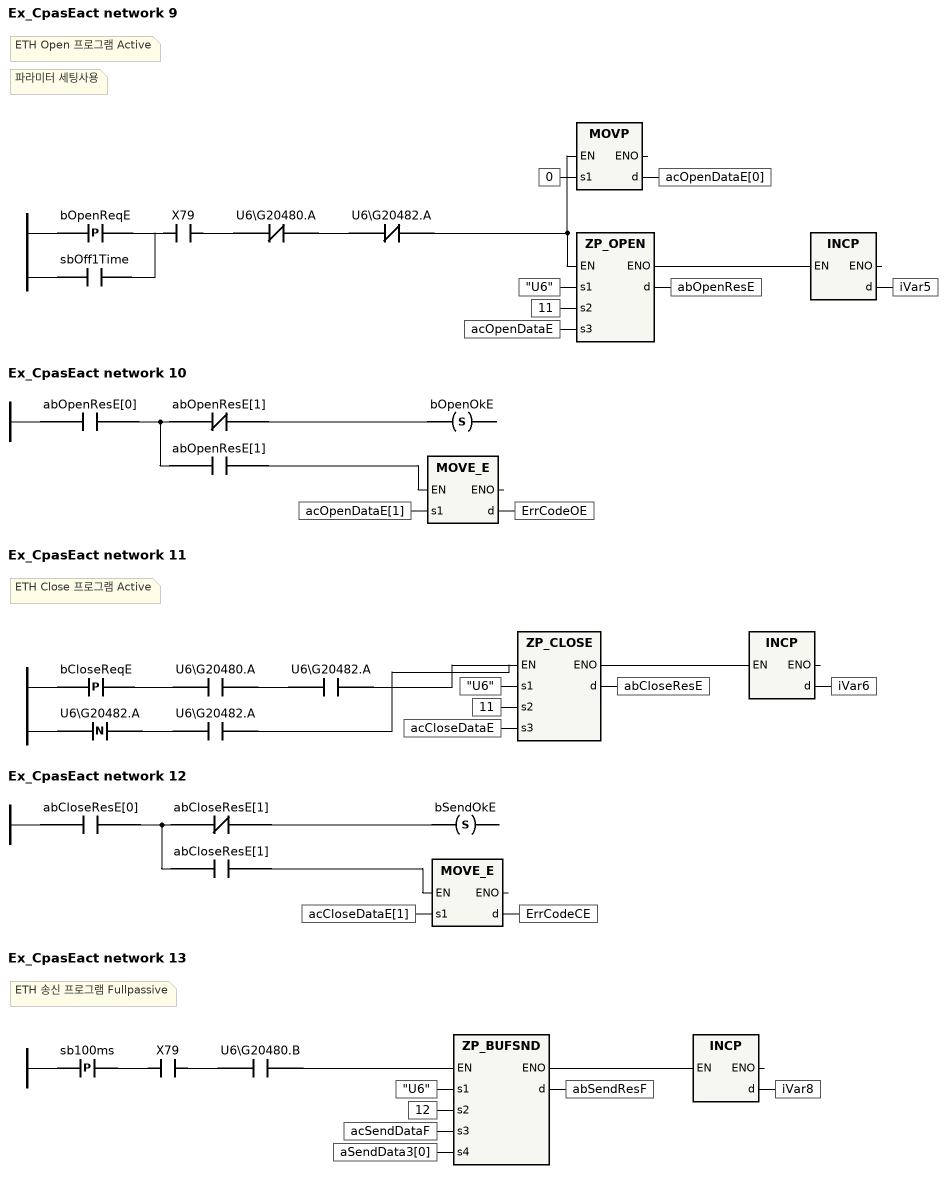
(* [picture p24: structured ladder/FBD of Ex_CpasEact, networks 9 to 13] *)
(* network 9 *)
(* ETH Open 프로그램 Active *)
(* 파라미터 세팅사용 *)
_p1 := (((LDP(TRUE, bOpenReqE) OR sbOff1Time) AND X79) AND NOT U6\G20480.A) AND NOT U6\G20482.A;
MOVP(_p1, 0, acOpenDataE[0]);
_e2 := ZP_OPEN(_p1, "U6", 11, acOpenDataE, abOpenResE);
INCP(_e2, iVar5);
(* network 10 *)
SET(abOpenResE[0] AND NOT abOpenResE[1], bOpenOkE);
MOVE_E(abOpenResE[0] AND abOpenResE[1], acOpenDataE[1], ErrCodeOE);
(* network 11 *)
(* ETH Close 프로그램 Active *)
_e1 := ZP_CLOSE((LDP(TRUE, bCloseReqE) AND U6\G20480.A AND U6\G20482.A) OR (LDF(TRUE, U6\G20482.A) AND U6\G20482.A), "U6", 11, acCloseDataE, abCloseResE);
INCP(_e1, iVar6);
(* network 12 *)
SET(abCloseResE[0] AND NOT abCloseResE[1], bSendOkE);
MOVE_E(abCloseResE[0] AND abCloseResE[1], acCloseDataE[1], ErrCodeCE);
(* network 13 *)
(* ETH 송신 프로그램 Fullpassive *)
_e1 := ZP_BUFSND(LDP(TRUE, sb100ms) AND X79 AND U6\G20480.B, "U6", 12, acSendDataF, aSendData3[0], abSendResF);
INCP(_e1, iVar8);
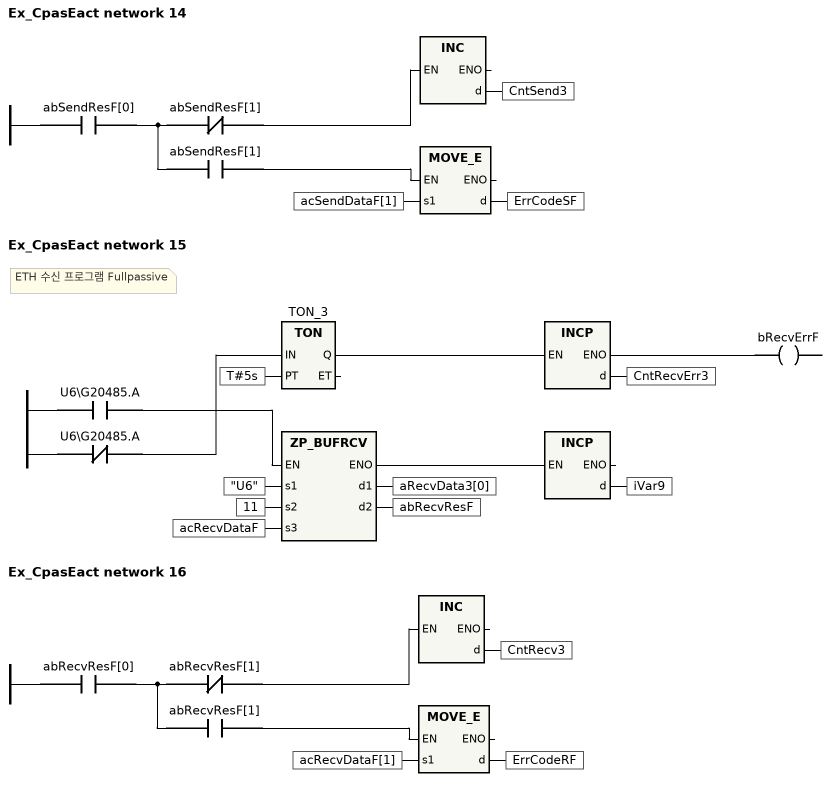
(* network 14 *)
INC(abSendResF[0] AND NOT abSendResF[1], CntSend3);
MOVE_E(abSendResF[0] AND abSendResF[1], acSendDataF[1], ErrCodeSF);
(* network 15 *)
(* ETH 수신 프로그램 Fullpassive *)
_e1 := ZP_BUFRCV(U6\G20485.A, "U6", 11, acRecvDataF, aRecvData3[0], abRecvResF);
INCP(_e1, iVar9);
TON_3(IN := NOT U6\G20485.A, PT := T#5s);
_e2 := INCP(TON_3.Q, CntRecvErr3);
bRecvErrF := _e2;
(* network 16 *)
INC(abRecvResF[0] AND NOT abRecvResF[1], CntRecv3);
MOVE_E(abRecvResF[0] AND abRecvResF[1], acRecvDataF[1], ErrCodeRF);
END_PROGRAM

PROGRAM Ex_SOCOPEN
VAR
  bOpenReqC : BOOL;
  bCsetReq : BOOL;
  bOpenReqE : BOOL;
  bOpenOkC : BOOL;
  bOpenOkE : BOOL;
  bOpenErrC : BOOL;
  bOpenErrE : BOOL;
  abOpenResC : ARRAY [0..1] OF BOOL;
  abOpenResE : ARRAY [0..1] OF BOOL;
  acOpenData : ARRAY [0..9] OF INT;
  acCsetData : ARRAY [0..4] OF INT;
  acRdCtrl : ARRAY [0..9] OF INT;
  bSendReqC : BOOL;
  bSendReqE : BOOL;
  bSendOkC : BOOL;
  bSendOkE : BOOL;
  bSendErrC : BOOL;
  bSendErrE : BOOL;
  abSendResC : ARRAY [0..1] OF BOOL;
  abSendResE : ARRAY [0..1] OF BOOL;
  abSendResF : ARRAY [0..1] OF BOOL;
  acSendDataC : ARRAY [0..1] OF INT;
  acSendDataE : ARRAY [0..1] OF INT;
  acSendDataF : ARRAY [0..1] OF INT;
  bRecvOkC : BOOL;
  bRecvOkE : BOOL;
  bRecvOkF : BOOL;
  bRecvErrC : BOOL;
  bRecvErrE : BOOL;
  bRecvErrF : BOOL;
  abRecvResC : ARRAY [0..1] OF BOOL;
  abRecvResE : ARRAY [0..1] OF BOOL;
  abRecvResF : ARRAY [0..1] OF BOOL;
  acRecvDataC : ARRAY [0..1] OF INT;
  acRecvDataE : ARRAY [0..1] OF INT;
  acRecvDataF : ARRAY [0..1] OF INT;
  bCloseReq : BOOL;
  bCloseOkC : BOOL;
  bCloseOkE : BOOL;
  bCloseErrC : BOOL;
  bCloseErrE : BOOL;
  abCloseResC : ARRAY [0..1] OF BOOL;
  abCloseResE : ARRAY [0..1] OF BOOL;
  acCloseData : ARRAY [0..1] OF INT;
  CntSend1 : INT;
  CntSend2 : INT;
  CntSend3 : INT;
  CntRecv1 : INT;
  CntRecvErr1 : INT;
  CntRecv2 : INT;
  CntRecv3 : INT;
  CntRecvErr2 : INT;
  CntRecvErr3 : INT;
  ErrCodeSC : INT;
  ErrCodeSE : INT;
  ErrCodeSF : INT;
  ErrCodeRC : INT;
  ErrCodeRE : INT;
  ErrCodeRF : INT;
  Mov4INT_1 : Mov4INT;
  Mov8INT_1 : Mov8INT;
  Mov4INT_2 : Mov4INT;
  Mov4INT_3 : Mov4INT;
  Mov4INT_4 : Mov4INT;
  Word2Bit8_1 : Word2Bit8;
  Word2Bit8_2 : Word2Bit8;
  Word2Bit8_3 : Word2Bit8;
  Word2Bit8_4 : Word2Bit8;
  Word2Bit8_5 : Word2Bit8;
  Word2Bit8_6 : Word2Bit8;
  TON_1 : TON;
  TON_2 : TON;
  TON_3 : TON;
END_VAR
(* structured ladder/FBD written out as ST: instructions are called as NAME(EN, inputs, outputs); _pN, _eN, _tN stand for wires *)
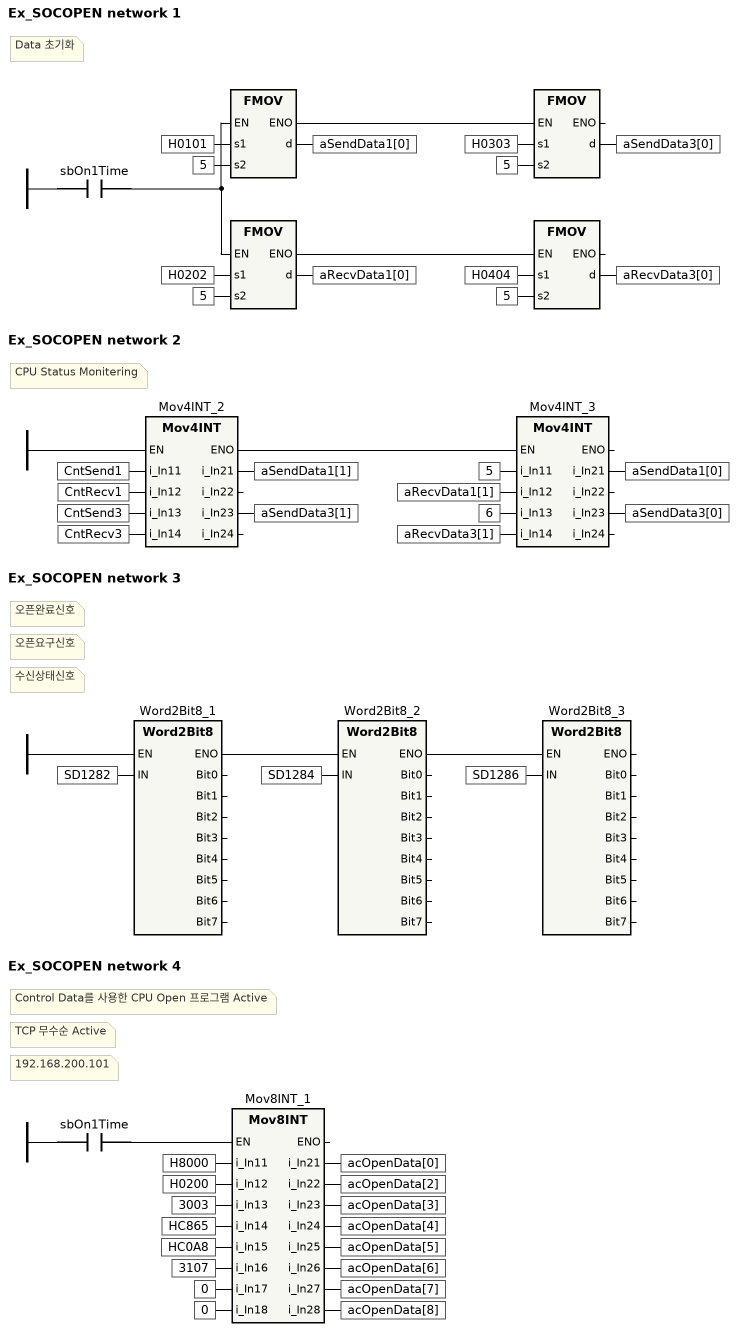
(* network 1 *)
(* Data 초기화 *)
_e1 := FMOV(sbOn1Time, H0101, 5, aSendData1[0]);
FMOV(_e1, H0303, 5, aSendData3[0]);
_e2 := FMOV(sbOn1Time, H0202, 5, aRecvData1[0]);
FMOV(_e2, H0404, 5, aRecvData3[0]);
(* network 2 *)
(* CPU Status Monitering *)
Mov4INT_2(EN := TRUE, i_In11 := CntSend1, i_In12 := CntRecv1, i_In13 := CntSend3, i_In14 := CntRecv3, i_In21 => aSendData1[1], i_In23 => aSendData3[1]);
Mov4INT_3(EN := Mov4INT_2.ENO, i_In11 := 5, i_In12 := aRecvData1[1], i_In13 := 6, i_In14 := aRecvData3[1], i_In21 => aSendData1[0], i_In23 => aSendData3[0]);
(* network 3 *)
(* 오픈완료신호 *)
(* 오픈요구신호 *)
(* 수신상태신호 *)
Word2Bit8_1(EN := TRUE, IN := SD1282);
Word2Bit8_2(EN := Word2Bit8_1.ENO, IN := SD1284);
Word2Bit8_3(EN := Word2Bit8_2.ENO, IN := SD1286);
(* network 4 *)
(* Control Data를 사용한 CPU Open 프로그램 Active *)
(* TCP 무수순 Active *)
(* 192.168.200.101 *)
Mov8INT_1(EN := sbOn1Time, i_In11 := H8000, i_In12 := H0200, i_In13 := 3003, i_In14 := HC865, i_In15 := HC0A8, i_In16 := 3107, i_In17 := 0, i_In18 := 0, i_In21 => acOpenData[0], i_In22 => acOpenData[2], i_In23 => acOpenData[3], i_In24 => acOpenData[4], i_In25 => acOpenData[5], i_In26 => acOpenData[6], i_In27 => acOpenData[7], i_In28 => acOpenData[8]);
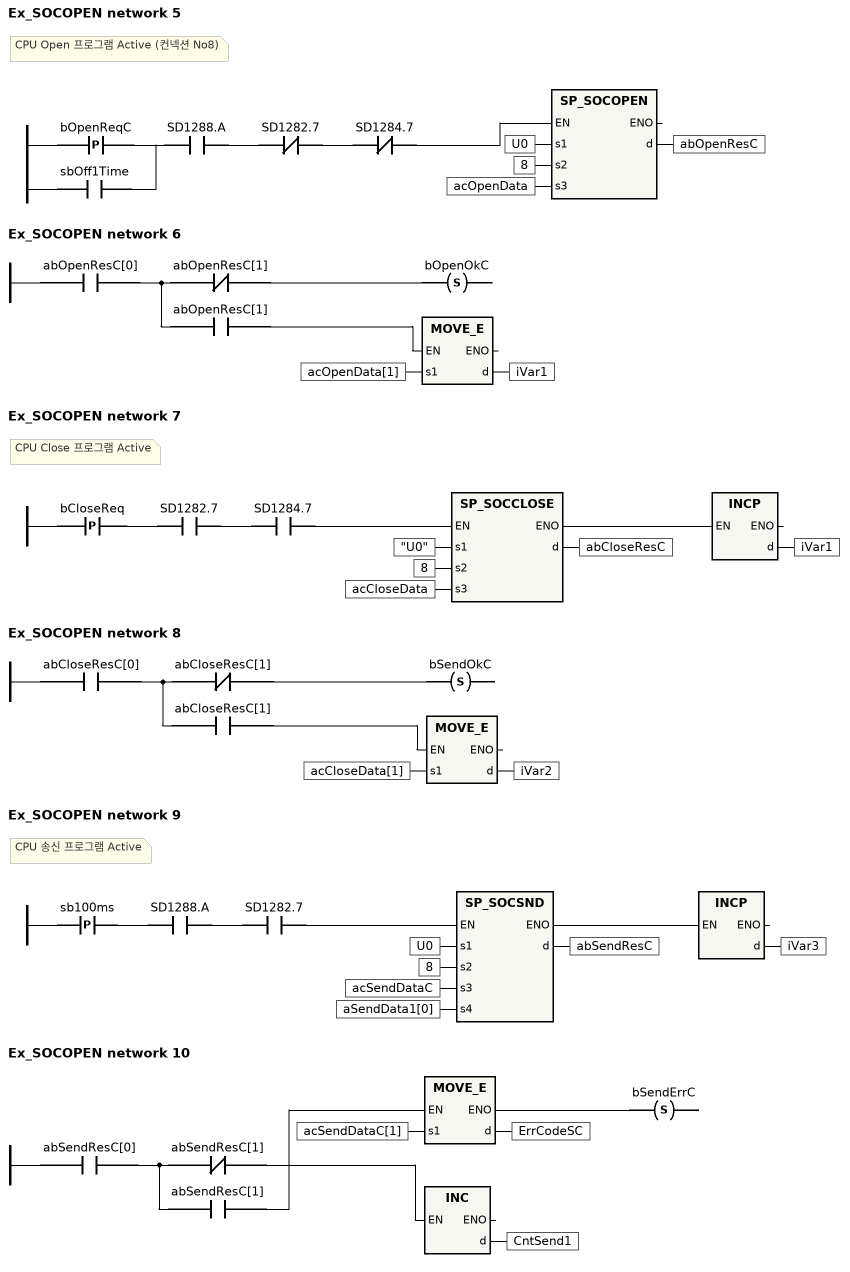
(* network 5 *)
(* CPU Open 프로그램 Active (컨넥션 No8) *)
SP_SOCOPEN((((LDP(TRUE, bOpenReqC) OR sbOff1Time) AND SD1288.A) AND NOT SD1282.7) AND NOT SD1284.7, U0, 8, acOpenData, abOpenResC);
(* network 6 *)
SET(abOpenResC[0] AND NOT abOpenResC[1], bOpenOkC);
MOVE_E(abOpenResC[0] AND abOpenResC[1], acOpenData[1], iVar1);
(* network 7 *)
(* CPU Close 프로그램 Active *)
_e1 := SP_SOCCLOSE(LDP(TRUE, bCloseReq) AND SD1282.7 AND SD1284.7, "U0", 8, acCloseData, abCloseResC);
INCP(_e1, iVar1);
(* network 8 *)
SET(abCloseResC[0] AND NOT abCloseResC[1], bSendOkC);
MOVE_E(abCloseResC[0] AND abCloseResC[1], acCloseData[1], iVar2);
(* network 9 *)
(* CPU 송신 프로그램 Active *)
_e1 := SP_SOCSND(LDP(TRUE, sb100ms) AND SD1288.A AND SD1282.7, U0, 8, acSendDataC, aSendData1[0], abSendResC);
INCP(_e1, iVar3);
(* network 10 *)
INC(abSendResC[0] AND NOT abSendResC[1], CntSend1);
_e1 := MOVE_E(abSendResC[0] AND abSendResC[1], acSendDataC[1], ErrCodeSC);
SET(_e1, bSendErrC);
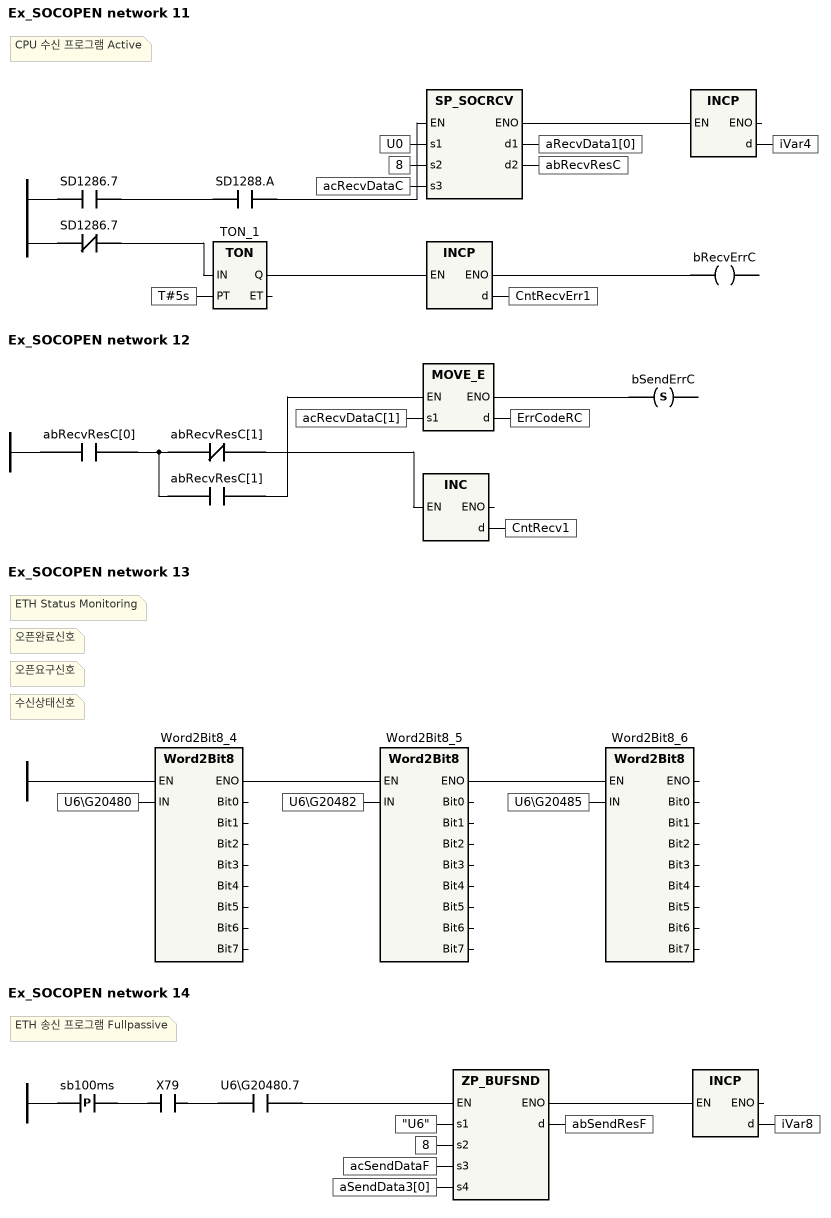
(* network 11 *)
(* CPU 수신 프로그램 Active *)
_e1 := SP_SOCRCV(SD1286.7 AND SD1288.A, U0, 8, acRecvDataC, aRecvData1[0], abRecvResC);
INCP(_e1, iVar4);
TON_1(IN := NOT SD1286.7, PT := T#5s);
_e2 := INCP(TON_1.Q, CntRecvErr1);
bRecvErrC := _e2;
(* network 12 *)
INC(abRecvResC[0] AND NOT abRecvResC[1], CntRecv1);
_e1 := MOVE_E(abRecvResC[0] AND abRecvResC[1], acRecvDataC[1], ErrCodeRC);
SET(_e1, bSendErrC);
(* network 13 *)
(* ETH Status Monitoring *)
(* 오픈완료신호 *)
(* 오픈요구신호 *)
(* 수신상태신호 *)
Word2Bit8_4(EN := TRUE, IN := U6\G20480);
Word2Bit8_5(EN := Word2Bit8_4.ENO, IN := U6\G20482);
Word2Bit8_6(EN := Word2Bit8_5.ENO, IN := U6\G20485);
(* network 14 *)
(* ETH 송신 프로그램 Fullpassive *)
_e1 := ZP_BUFSND(LDP(TRUE, sb100ms) AND X79 AND U6\G20480.7, "U6", 8, acSendDataF, aSendData3[0], abSendResF);
INCP(_e1, iVar8);
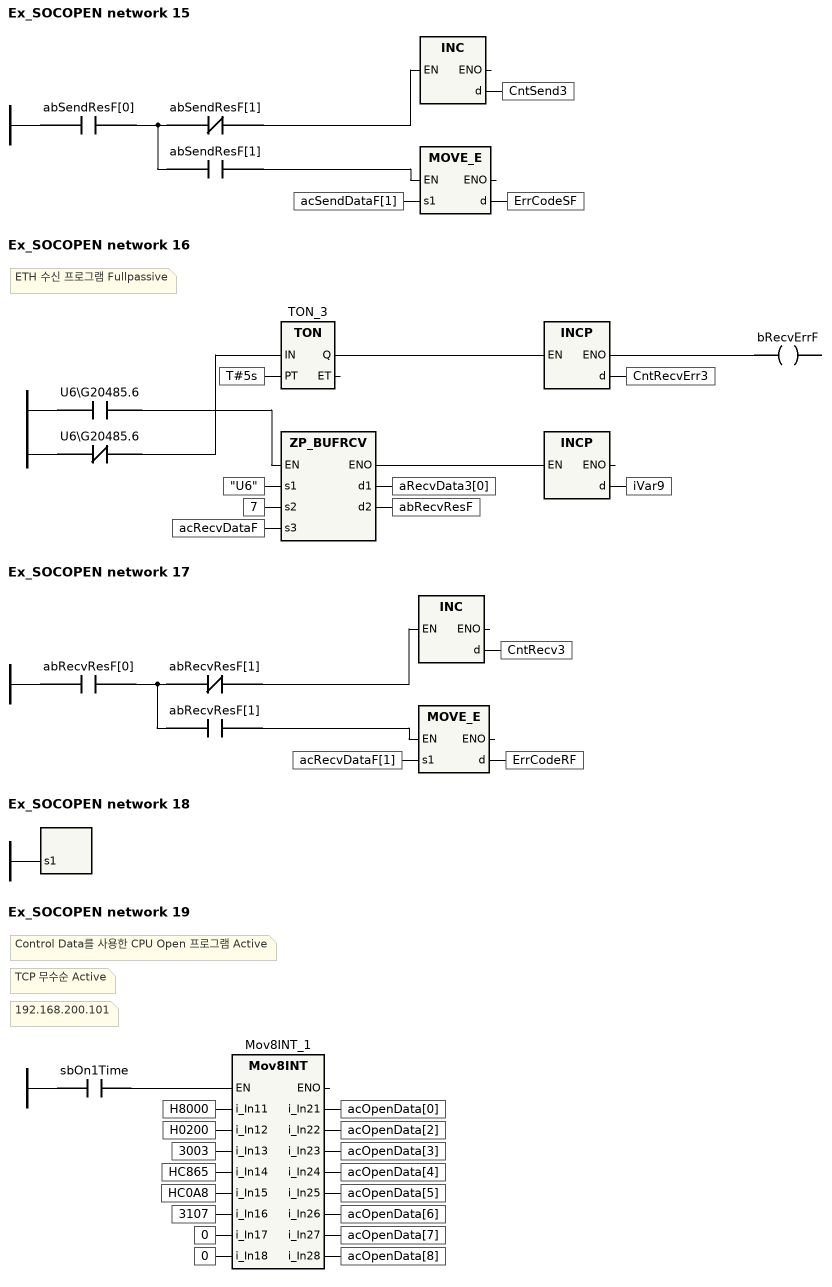
(* network 15 *)
INC(abSendResF[0] AND NOT abSendResF[1], CntSend3);
MOVE_E(abSendResF[0] AND abSendResF[1], acSendDataF[1], ErrCodeSF);
(* network 16 *)
(* ETH 수신 프로그램 Fullpassive *)
_e1 := ZP_BUFRCV(U6\G20485.6, "U6", 7, acRecvDataF, aRecvData3[0], abRecvResF);
INCP(_e1, iVar9);
TON_3(IN := NOT U6\G20485.6, PT := T#5s);
_e2 := INCP(TON_3.Q, CntRecvErr3);
bRecvErrF := _e2;
(* network 17 *)
INC(abRecvResF[0] AND NOT abRecvResF[1], CntRecv3);
MOVE_E(abRecvResF[0] AND abRecvResF[1], acRecvDataF[1], ErrCodeRF);
(* network 18 *)
(* element kind 10  <- TRUE *)
(* network 19 *)
(* Control Data를 사용한 CPU Open 프로그램 Active *)
(* TCP 무수순 Active *)
(* 192.168.200.101 *)
Mov8INT_1(EN := sbOn1Time, i_In11 := H8000, i_In12 := H0200, i_In13 := 3003, i_In14 := HC865, i_In15 := HC0A8, i_In16 := 3107, i_In17 := 0, i_In18 := 0, i_In21 => acOpenData[0], i_In22 => acOpenData[2], i_In23 => acOpenData[3], i_In24 => acOpenData[4], i_In25 => acOpenData[5], i_In26 => acOpenData[6], i_In27 => acOpenData[7], i_In28 => acOpenData[8]);
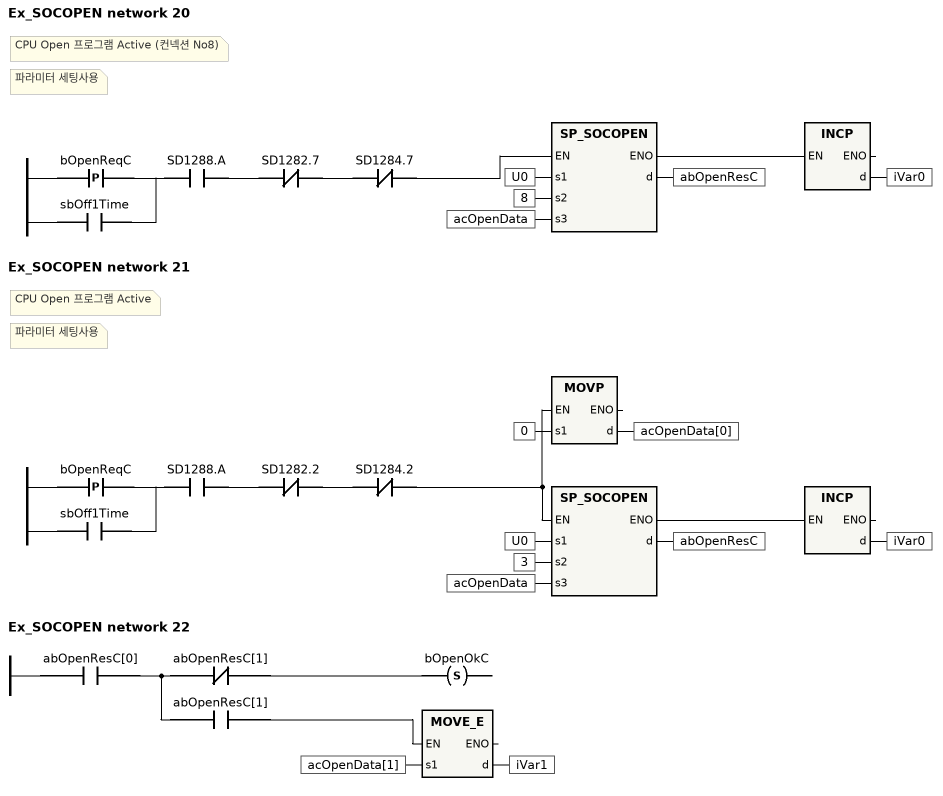
(* network 20 *)
(* CPU Open 프로그램 Active (컨넥션 No8) *)
(* 파라미터 세팅사용 *)
_e1 := SP_SOCOPEN((((LDP(TRUE, bOpenReqC) OR sbOff1Time) AND SD1288.A) AND NOT SD1282.7) AND NOT SD1284.7, U0, 8, acOpenData, abOpenResC);
INCP(_e1, iVar0);
(* network 21 *)
(* CPU Open 프로그램 Active *)
(* 파라미터 세팅사용 *)
_p1 := (((LDP(TRUE, bOpenReqC) OR sbOff1Time) AND SD1288.A) AND NOT SD1282.2) AND NOT SD1284.2;
MOVP(_p1, 0, acOpenData[0]);
_e2 := SP_SOCOPEN(_p1, U0, 3, acOpenData, abOpenResC);
INCP(_e2, iVar0);
(* network 22 *)
SET(abOpenResC[0] AND NOT abOpenResC[1], bOpenOkC);
MOVE_E(abOpenResC[0] AND abOpenResC[1], acOpenData[1], iVar1);
END_PROGRAM

PROGRAM Ex_SOCCLOSE
VAR
  bOpenReqC : BOOL;
  bCsetReq : BOOL;
  bOpenReqE : BOOL;
  bOpenOkC : BOOL;
  bOpenOkE : BOOL;
  bOpenErrC : BOOL;
  bOpenErrE : BOOL;
  abOpenResC : ARRAY [0..1] OF BOOL;
  abOpenResE : ARRAY [0..1] OF BOOL;
  acOpenData : ARRAY [0..9] OF INT;
  acCsetData : ARRAY [0..4] OF INT;
  acRdCtrl : ARRAY [0..9] OF INT;
  bSendReqC : BOOL;
  bSendReqE : BOOL;
  bSendOkC : BOOL;
  bSendOkE : BOOL;
  bSendErrC : BOOL;
  bSendErrE : BOOL;
  abSendResC : ARRAY [0..1] OF BOOL;
  abSendResE : ARRAY [0..1] OF BOOL;
  abSendResF : ARRAY [0..1] OF BOOL;
  acSendDataC : ARRAY [0..1] OF INT;
  acSendDataE : ARRAY [0..1] OF INT;
  acSendDataF : ARRAY [0..1] OF INT;
  bRecvOkC : BOOL;
  bRecvOkE : BOOL;
  bRecvOkF : BOOL;
  bRecvErrC : BOOL;
  bRecvErrE : BOOL;
  bRecvErrF : BOOL;
  abRecvResC : ARRAY [0..1] OF BOOL;
  abRecvResE : ARRAY [0..1] OF BOOL;
  abRecvResF : ARRAY [0..1] OF BOOL;
  acRecvDataC : ARRAY [0..1] OF INT;
  acRecvDataE : ARRAY [0..1] OF INT;
  acRecvDataF : ARRAY [0..1] OF INT;
  bCloseReq : BOOL;
  bCloseOkC : BOOL;
  bCloseOkE : BOOL;
  bCloseErrC : BOOL;
  bCloseErrE : BOOL;
  abCloseResC : ARRAY [0..1] OF BOOL;
  abCloseResE : ARRAY [0..1] OF BOOL;
  acCloseData : ARRAY [0..1] OF INT;
  CntSend1 : INT;
  CntSend2 : INT;
  CntSend3 : INT;
  CntRecv1 : INT;
  CntRecvErr1 : INT;
  CntRecv2 : INT;
  CntRecv3 : INT;
  CntRecvErr2 : INT;
  CntRecvErr3 : INT;
  ErrCodeSC : INT;
  ErrCodeSE : INT;
  ErrCodeSF : INT;
  ErrCodeRC : INT;
  ErrCodeRE : INT;
  ErrCodeRF : INT;
  Mov4INT_1 : Mov4INT;
  Mov8INT_1 : Mov8INT;
  Mov4INT_2 : Mov4INT;
  Mov4INT_3 : Mov4INT;
  Mov4INT_4 : Mov4INT;
  Word2Bit8_1 : Word2Bit8;
  Word2Bit8_2 : Word2Bit8;
  Word2Bit8_3 : Word2Bit8;
  Word2Bit8_4 : Word2Bit8;
  Word2Bit8_5 : Word2Bit8;
  Word2Bit8_6 : Word2Bit8;
  TON_1 : TON;
  TON_2 : TON;
  TON_3 : TON;
  bFlag : BOOL;
  bFlagExe : BOOL;
  bNormal : BOOL;
  bError : BOOL;
END_VAR
(* structured ladder/FBD written out as ST: instructions are called as NAME(EN, inputs, outputs); _pN, _eN, _tN stand for wires *)
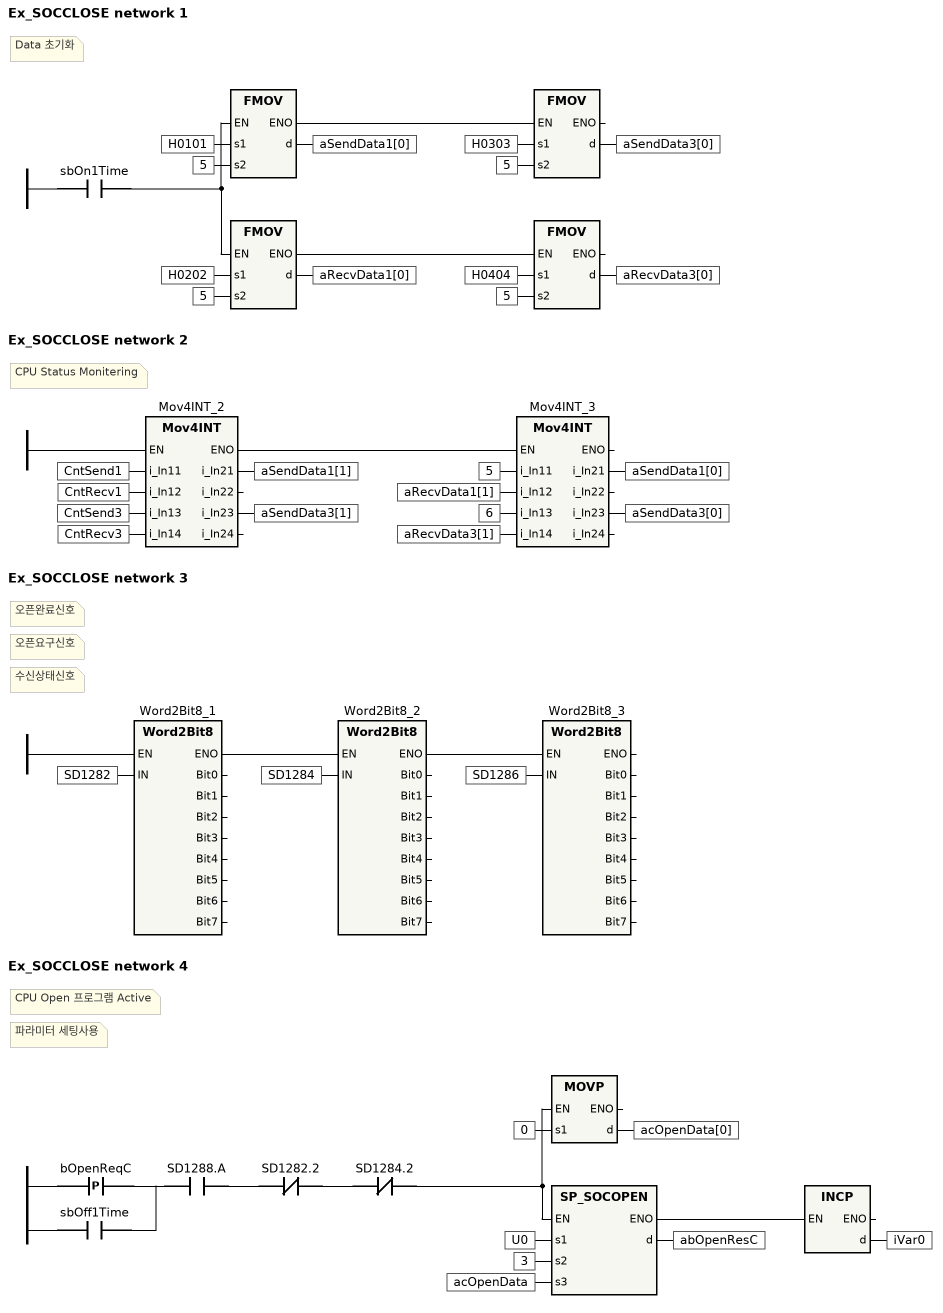
(* network 1 *)
(* Data 초기화 *)
_e1 := FMOV(sbOn1Time, H0101, 5, aSendData1[0]);
FMOV(_e1, H0303, 5, aSendData3[0]);
_e2 := FMOV(sbOn1Time, H0202, 5, aRecvData1[0]);
FMOV(_e2, H0404, 5, aRecvData3[0]);
(* network 2 *)
(* CPU Status Monitering *)
Mov4INT_2(EN := TRUE, i_In11 := CntSend1, i_In12 := CntRecv1, i_In13 := CntSend3, i_In14 := CntRecv3, i_In21 => aSendData1[1], i_In23 => aSendData3[1]);
Mov4INT_3(EN := Mov4INT_2.ENO, i_In11 := 5, i_In12 := aRecvData1[1], i_In13 := 6, i_In14 := aRecvData3[1], i_In21 => aSendData1[0], i_In23 => aSendData3[0]);
(* network 3 *)
(* 오픈완료신호 *)
(* 오픈요구신호 *)
(* 수신상태신호 *)
Word2Bit8_1(EN := TRUE, IN := SD1282);
Word2Bit8_2(EN := Word2Bit8_1.ENO, IN := SD1284);
Word2Bit8_3(EN := Word2Bit8_2.ENO, IN := SD1286);
(* network 4 *)
(* CPU Open 프로그램 Active *)
(* 파라미터 세팅사용 *)
_p1 := (((LDP(TRUE, bOpenReqC) OR sbOff1Time) AND SD1288.A) AND NOT SD1282.2) AND NOT SD1284.2;
MOVP(_p1, 0, acOpenData[0]);
_e2 := SP_SOCOPEN(_p1, U0, 3, acOpenData, abOpenResC);
INCP(_e2, iVar0);
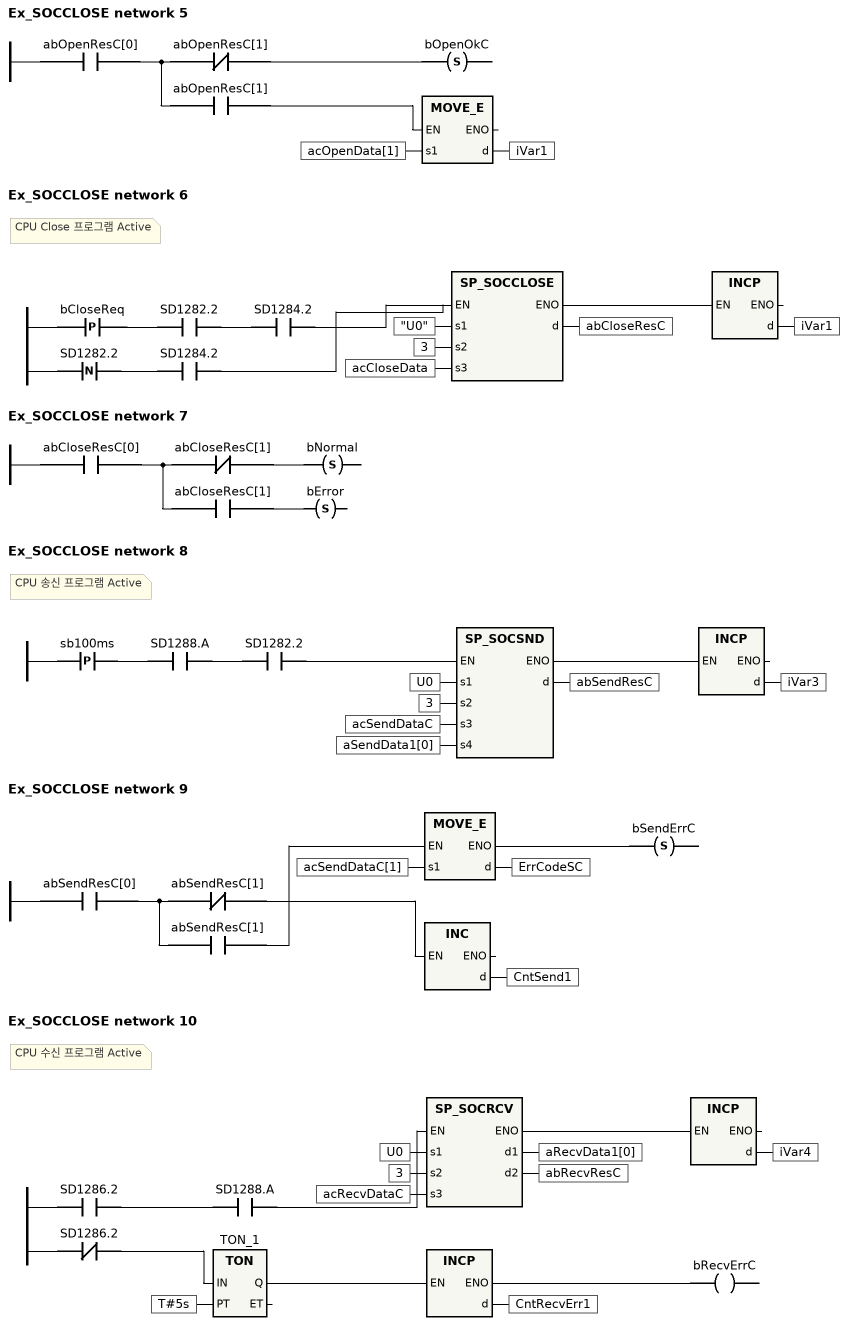
(* network 5 *)
SET(abOpenResC[0] AND NOT abOpenResC[1], bOpenOkC);
MOVE_E(abOpenResC[0] AND abOpenResC[1], acOpenData[1], iVar1);
(* network 6 *)
(* CPU Close 프로그램 Active *)
_e1 := SP_SOCCLOSE((LDP(TRUE, bCloseReq) AND SD1282.2 AND SD1284.2) OR (LDF(TRUE, SD1282.2) AND SD1284.2), "U0", 3, acCloseData, abCloseResC);
INCP(_e1, iVar1);
(* network 7 *)
SET(abCloseResC[0] AND NOT abCloseResC[1], bNormal);
SET(abCloseResC[0] AND abCloseResC[1], bError);
(* network 8 *)
(* CPU 송신 프로그램 Active *)
_e1 := SP_SOCSND(LDP(TRUE, sb100ms) AND SD1288.A AND SD1282.2, U0, 3, acSendDataC, aSendData1[0], abSendResC);
INCP(_e1, iVar3);
(* network 9 *)
INC(abSendResC[0] AND NOT abSendResC[1], CntSend1);
_e1 := MOVE_E(abSendResC[0] AND abSendResC[1], acSendDataC[1], ErrCodeSC);
SET(_e1, bSendErrC);
(* network 10 *)
(* CPU 수신 프로그램 Active *)
_e1 := SP_SOCRCV(SD1286.2 AND SD1288.A, U0, 3, acRecvDataC, aRecvData1[0], abRecvResC);
INCP(_e1, iVar4);
TON_1(IN := NOT SD1286.2, PT := T#5s);
_e2 := INCP(TON_1.Q, CntRecvErr1);
bRecvErrC := _e2;
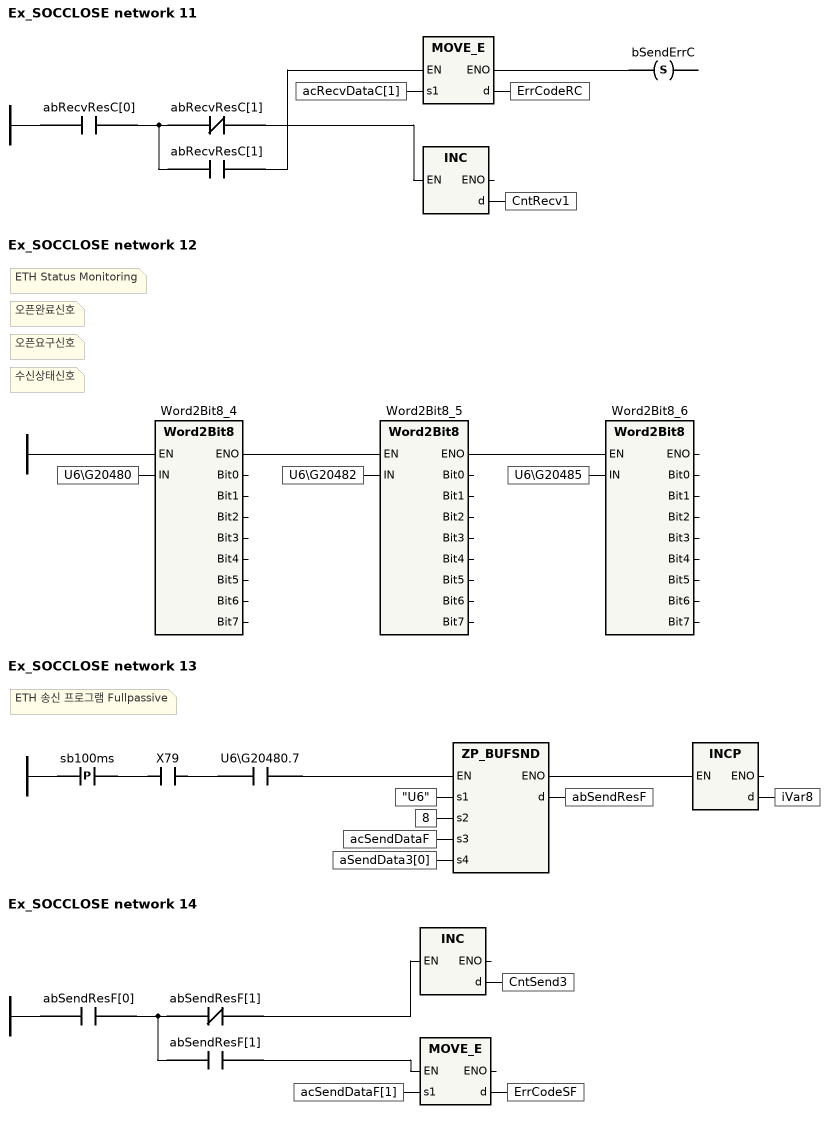
(* network 11 *)
INC(abRecvResC[0] AND NOT abRecvResC[1], CntRecv1);
_e1 := MOVE_E(abRecvResC[0] AND abRecvResC[1], acRecvDataC[1], ErrCodeRC);
SET(_e1, bSendErrC);
(* network 12 *)
(* ETH Status Monitoring *)
(* 오픈완료신호 *)
(* 오픈요구신호 *)
(* 수신상태신호 *)
Word2Bit8_4(EN := TRUE, IN := U6\G20480);
Word2Bit8_5(EN := Word2Bit8_4.ENO, IN := U6\G20482);
Word2Bit8_6(EN := Word2Bit8_5.ENO, IN := U6\G20485);
(* network 13 *)
(* ETH 송신 프로그램 Fullpassive *)
_e1 := ZP_BUFSND(LDP(TRUE, sb100ms) AND X79 AND U6\G20480.7, "U6", 8, acSendDataF, aSendData3[0], abSendResF);
INCP(_e1, iVar8);
(* network 14 *)
INC(abSendResF[0] AND NOT abSendResF[1], CntSend3);
MOVE_E(abSendResF[0] AND abSendResF[1], acSendDataF[1], ErrCodeSF);
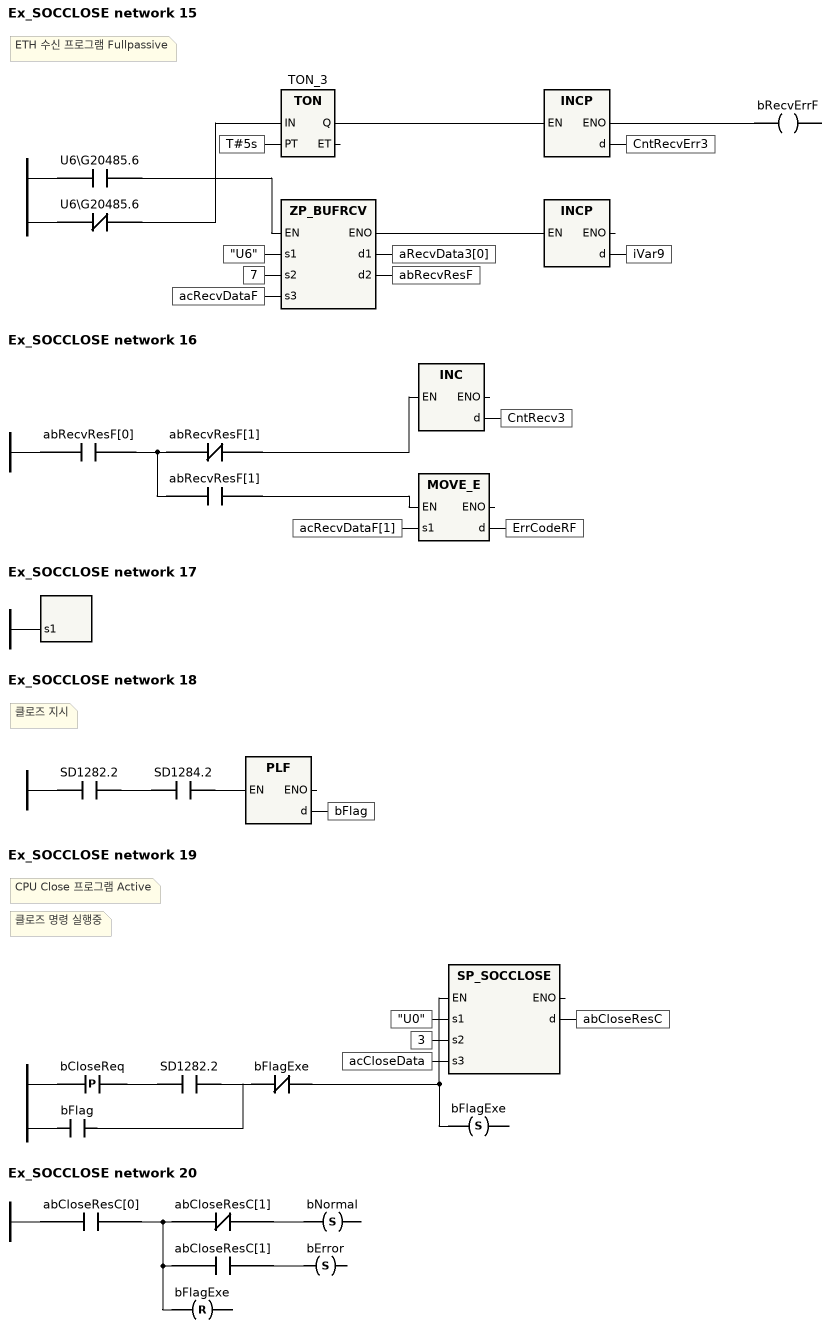
(* network 15 *)
(* ETH 수신 프로그램 Fullpassive *)
_e1 := ZP_BUFRCV(U6\G20485.6, "U6", 7, acRecvDataF, aRecvData3[0], abRecvResF);
INCP(_e1, iVar9);
TON_3(IN := NOT U6\G20485.6, PT := T#5s);
_e2 := INCP(TON_3.Q, CntRecvErr3);
bRecvErrF := _e2;
(* network 16 *)
INC(abRecvResF[0] AND NOT abRecvResF[1], CntRecv3);
MOVE_E(abRecvResF[0] AND abRecvResF[1], acRecvDataF[1], ErrCodeRF);
(* network 17 *)
(* element kind 10  <- TRUE *)
(* network 18 *)
(* 클로즈 지시 *)
PLF(SD1282.2 AND SD1284.2, bFlag);
(* network 19 *)
(* CPU Close 프로그램 Active *)
(* 클로즈 명령 실행중 *)
_p1 := ((LDP(TRUE, bCloseReq) AND SD1282.2) OR bFlag) AND NOT bFlagExe;
SP_SOCCLOSE(_p1, "U0", 3, acCloseData, abCloseResC);
SET(_p1, bFlagExe);
(* network 20 *)
SET(abCloseResC[0] AND NOT abCloseResC[1], bNormal);
SET(abCloseResC[0] AND abCloseResC[1], bError);
RST(abCloseResC[0], bFlagExe);
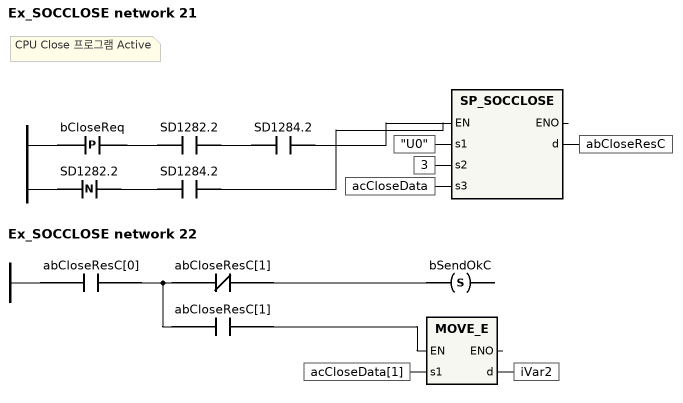
(* network 21 *)
(* CPU Close 프로그램 Active *)
SP_SOCCLOSE((LDP(TRUE, bCloseReq) AND SD1282.2 AND SD1284.2) OR (LDF(TRUE, SD1282.2) AND SD1284.2), "U0", 3, acCloseData, abCloseResC);
(* network 22 *)
SET(abCloseResC[0] AND NOT abCloseResC[1], bSendOkC);
MOVE_E(abCloseResC[0] AND abCloseResC[1], acCloseData[1], iVar2);
END_PROGRAM

PROGRAM Ex_SOCRCV
VAR
  bOpenReqC : BOOL;
  bOpenOkC : BOOL;
  bOpenErrC : BOOL;
  abOpenResC : ARRAY [0..1] OF BOOL;
  acOpenData : ARRAY [0..9] OF INT;
  bSendReqC : BOOL;
  bSendOkC : BOOL;
  bSendErrC : BOOL;
  abSendResC : ARRAY [0..1] OF BOOL;
  acSendDataC : ARRAY [0..1] OF INT;
  bRecvOkC : BOOL;
  bRecvErrC : BOOL;
  abRecvResC : ARRAY [0..1] OF BOOL;
  bCloseReq : BOOL;
  bCloseOkC : BOOL;
  bCloseErrC : BOOL;
  abCloseResC : ARRAY [0..1] OF BOOL;
  acCloseData : ARRAY [0..1] OF INT;
  CntSend1 : INT;
  CntSend2 : INT;
  CntRecv1 : INT;
  CntRecv2 : INT;
  Mov4INT_1 : Mov4INT;
  Mov8INT_1 : Mov8INT;
  acRdCtrl : ARRAY [0..9] OF INT;
  Mov4INT_2 : Mov4INT;
  bOpenReqE : BOOL;
  bOpenOkE : BOOL;
  bOpenErrE : BOOL;
  abOpenResE : ARRAY [0..1] OF BOOL;
  bSendErrE : BOOL;
  bSendOkE : BOOL;
  bSendReqE : BOOL;
  abSendResE : ARRAY [0..1] OF BOOL;
  abRecvResE : ARRAY [0..1] OF BOOL;
  bRecvErrE : BOOL;
  bRecvOkE : BOOL;
  abCloseResE : ARRAY [0..1] OF BOOL;
  bCloseErrE : BOOL;
  bCloseOkE : BOOL;
  acSendDataE : ARRAY [0..1] OF INT;
  acRecvDataC : ARRAY [0..1] OF INT;
  acRecvDataE : ARRAY [0..1] OF INT;
  Word2Bit8_1 : Word2Bit8;
  Word2Bit8_2 : Word2Bit8;
  Word2Bit8_3 : Word2Bit8;
  Word2Bit8_4 : Word2Bit8;
  Word2Bit8_5 : Word2Bit8;
  Word2Bit8_6 : Word2Bit8;
  ErrCodeSC : INT;
  ErrCodeSE : INT;
  Mov4INT_3 : Mov4INT;
  bChangeReqC : BOOL;
  Mov4INT_4 : Mov4INT;
  acCsetData : ARRAY [0..4] OF INT;
  TON_1 : TON;
  CntRecvErr1 : INT;
  CntRecvErr2 : INT;
  TON_2 : TON;
  ErrCodeRC : INT;
  ErrCodeRE : INT;
END_VAR
(* structured ladder/FBD written out as ST: instructions are called as NAME(EN, inputs, outputs); _pN, _eN, _tN stand for wires *)
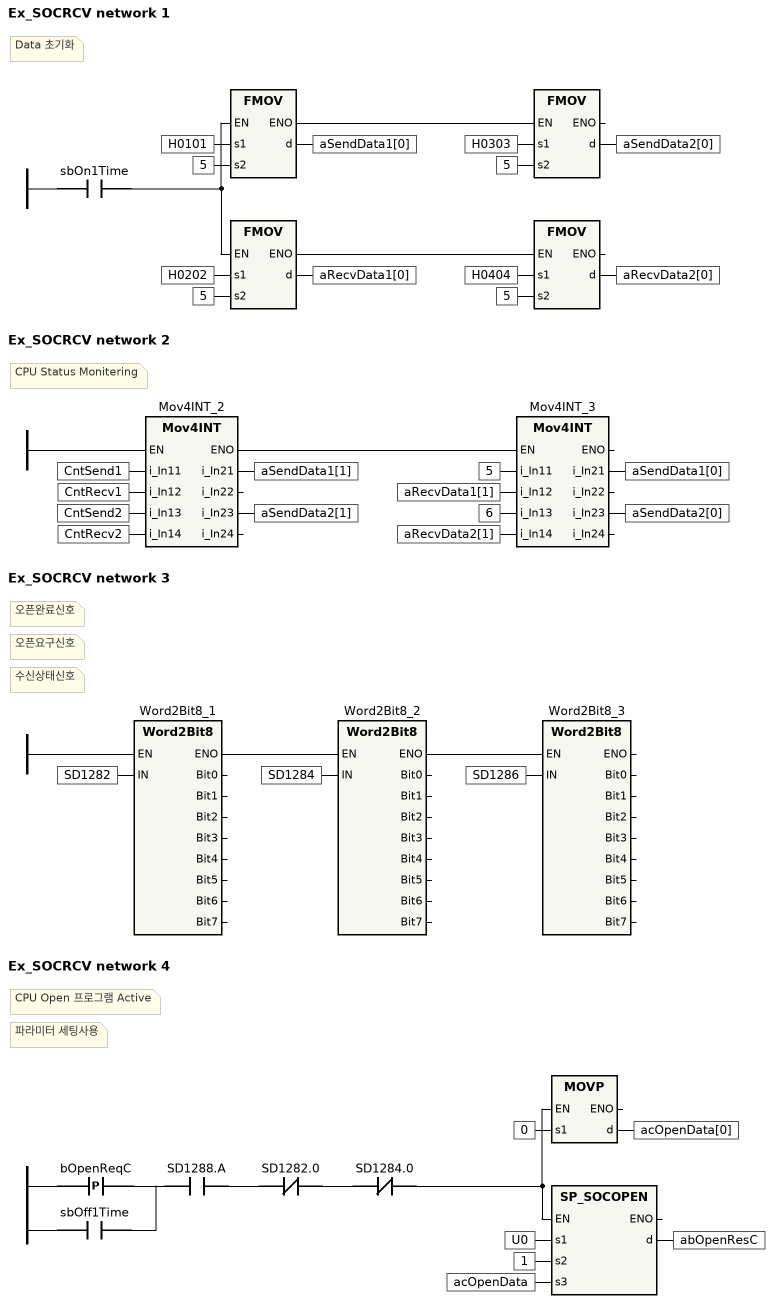
(* network 1 *)
(* Data 초기화 *)
_e1 := FMOV(sbOn1Time, H0101, 5, aSendData1[0]);
FMOV(_e1, H0303, 5, aSendData2[0]);
_e2 := FMOV(sbOn1Time, H0202, 5, aRecvData1[0]);
FMOV(_e2, H0404, 5, aRecvData2[0]);
(* network 2 *)
(* CPU Status Monitering *)
Mov4INT_2(EN := TRUE, i_In11 := CntSend1, i_In12 := CntRecv1, i_In13 := CntSend2, i_In14 := CntRecv2, i_In21 => aSendData1[1], i_In23 => aSendData2[1]);
Mov4INT_3(EN := Mov4INT_2.ENO, i_In11 := 5, i_In12 := aRecvData1[1], i_In13 := 6, i_In14 := aRecvData2[1], i_In21 => aSendData1[0], i_In23 => aSendData2[0]);
(* network 3 *)
(* 오픈완료신호 *)
(* 오픈요구신호 *)
(* 수신상태신호 *)
Word2Bit8_1(EN := TRUE, IN := SD1282);
Word2Bit8_2(EN := Word2Bit8_1.ENO, IN := SD1284);
Word2Bit8_3(EN := Word2Bit8_2.ENO, IN := SD1286);
(* network 4 *)
(* CPU Open 프로그램 Active *)
(* 파라미터 세팅사용 *)
_p1 := (((LDP(TRUE, bOpenReqC) OR sbOff1Time) AND SD1288.A) AND NOT SD1282.0) AND NOT SD1284.0;
MOVP(_p1, 0, acOpenData[0]);
SP_SOCOPEN(_p1, U0, 1, acOpenData, abOpenResC);
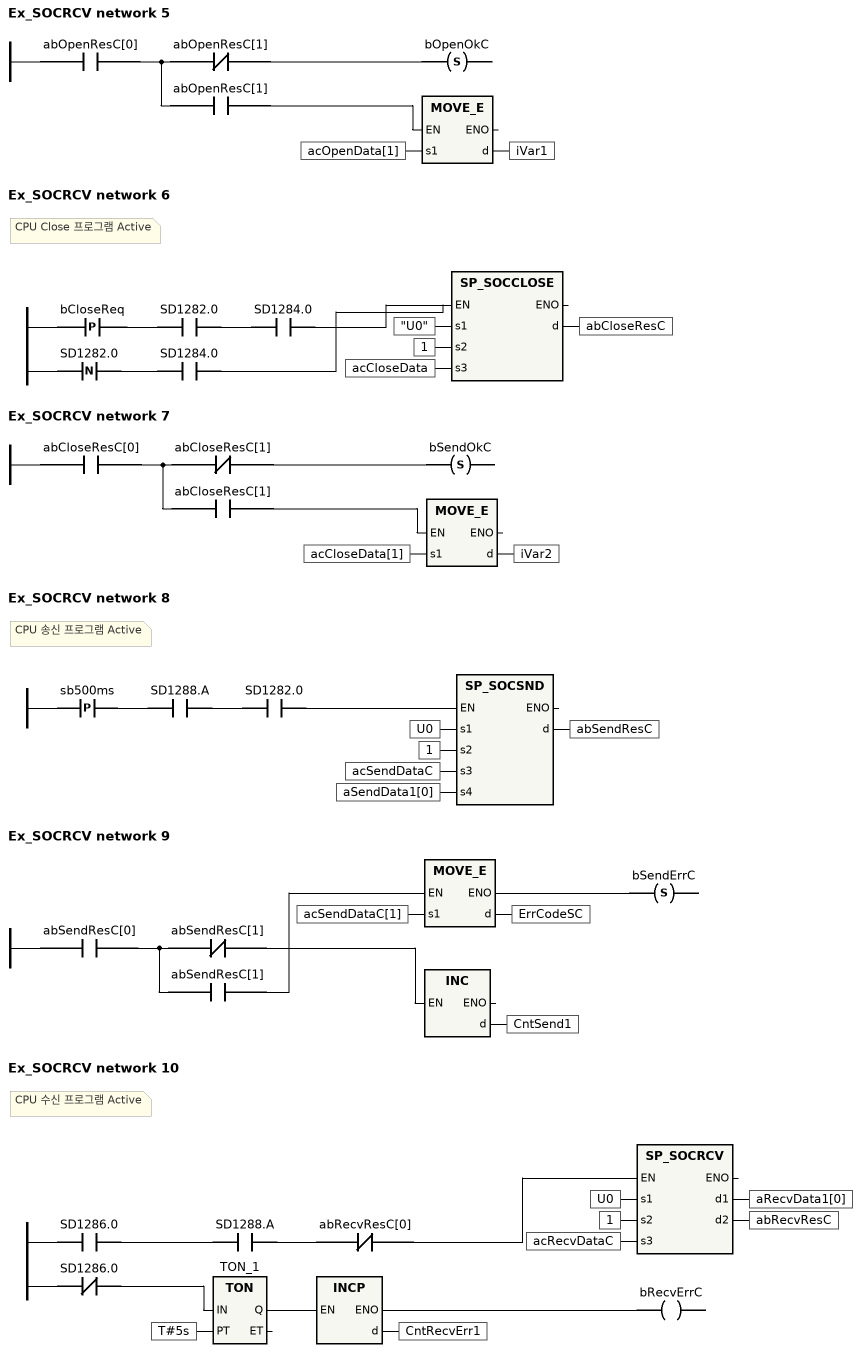
(* network 5 *)
SET(abOpenResC[0] AND NOT abOpenResC[1], bOpenOkC);
MOVE_E(abOpenResC[0] AND abOpenResC[1], acOpenData[1], iVar1);
(* network 6 *)
(* CPU Close 프로그램 Active *)
SP_SOCCLOSE((LDP(TRUE, bCloseReq) AND SD1282.0 AND SD1284.0) OR (LDF(TRUE, SD1282.0) AND SD1284.0), "U0", 1, acCloseData, abCloseResC);
(* network 7 *)
SET(abCloseResC[0] AND NOT abCloseResC[1], bSendOkC);
MOVE_E(abCloseResC[0] AND abCloseResC[1], acCloseData[1], iVar2);
(* network 8 *)
(* CPU 송신 프로그램 Active *)
SP_SOCSND(LDP(TRUE, sb500ms) AND SD1288.A AND SD1282.0, U0, 1, acSendDataC, aSendData1[0], abSendResC);
(* network 9 *)
INC(abSendResC[0] AND NOT abSendResC[1], CntSend1);
_e1 := MOVE_E(abSendResC[0] AND abSendResC[1], acSendDataC[1], ErrCodeSC);
SET(_e1, bSendErrC);
(* network 10 *)
(* CPU 수신 프로그램 Active *)
SP_SOCRCV(SD1286.0 AND SD1288.A AND NOT abRecvResC[0], U0, 1, acRecvDataC, aRecvData1[0], abRecvResC);
TON_1(IN := NOT SD1286.0, PT := T#5s);
_e1 := INCP(TON_1.Q, CntRecvErr1);
bRecvErrC := _e1;
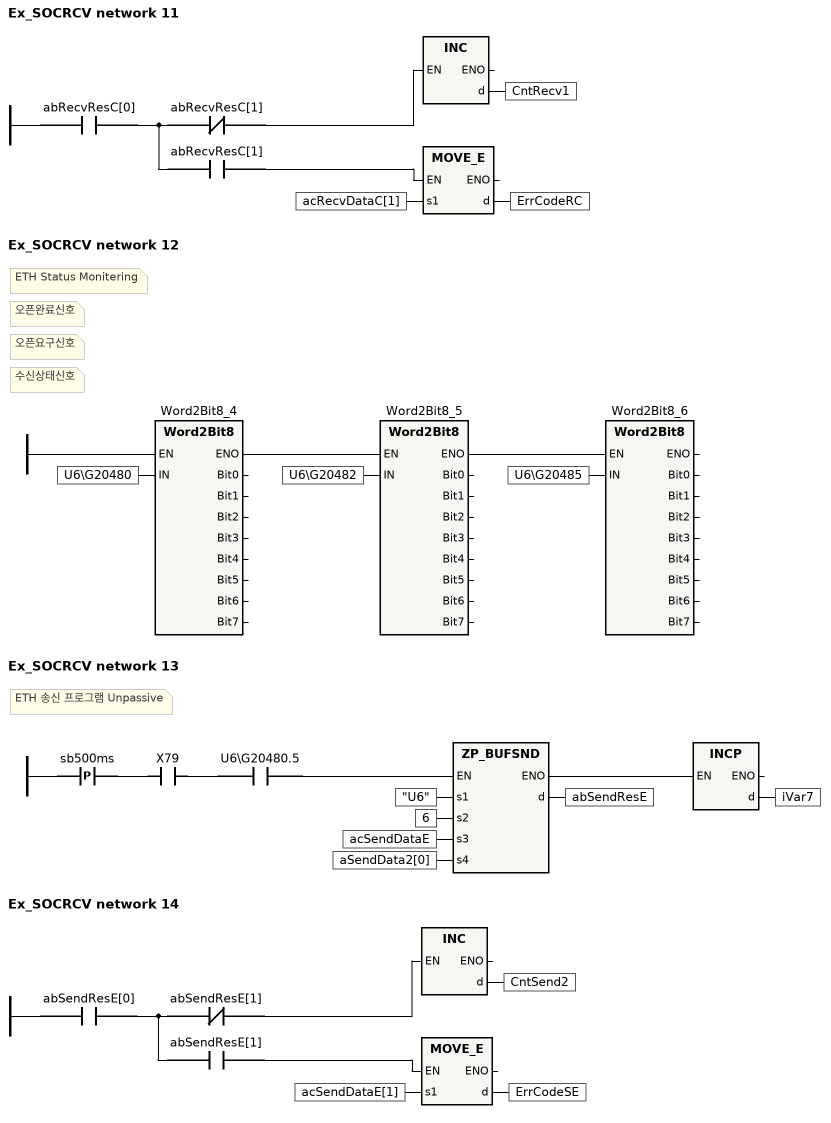
(* network 11 *)
INC(abRecvResC[0] AND NOT abRecvResC[1], CntRecv1);
MOVE_E(abRecvResC[0] AND abRecvResC[1], acRecvDataC[1], ErrCodeRC);
(* network 12 *)
(* ETH Status Monitering *)
(* 오픈완료신호 *)
(* 오픈요구신호 *)
(* 수신상태신호 *)
Word2Bit8_4(EN := TRUE, IN := U6\G20480);
Word2Bit8_5(EN := Word2Bit8_4.ENO, IN := U6\G20482);
Word2Bit8_6(EN := Word2Bit8_5.ENO, IN := U6\G20485);
(* network 13 *)
(* ETH 송신 프로그램 Unpassive *)
_e1 := ZP_BUFSND(LDP(TRUE, sb500ms) AND X79 AND U6\G20480.5, "U6", 6, acSendDataE, aSendData2[0], abSendResE);
INCP(_e1, iVar7);
(* network 14 *)
INC(abSendResE[0] AND NOT abSendResE[1], CntSend2);
MOVE_E(abSendResE[0] AND abSendResE[1], acSendDataE[1], ErrCodeSE);
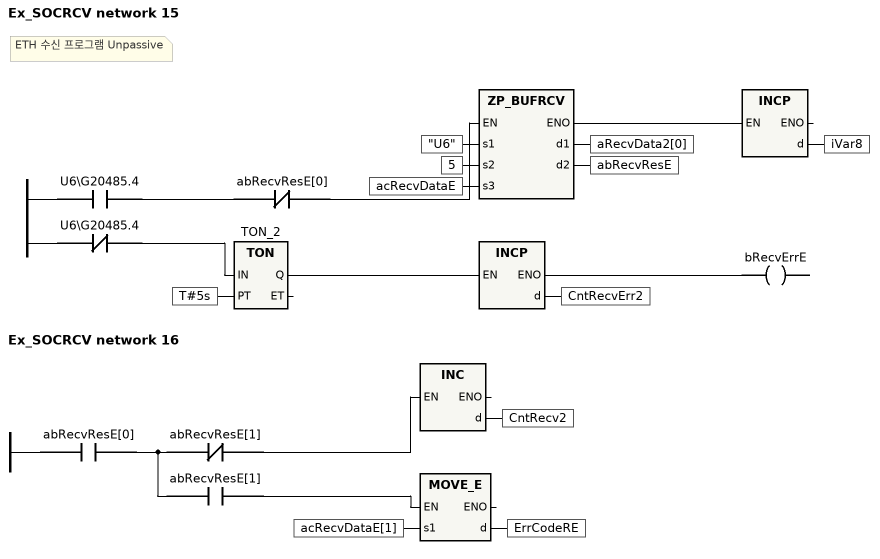
(* network 15 *)
(* ETH 수신 프로그램 Unpassive *)
_e1 := ZP_BUFRCV(U6\G20485.4 AND NOT abRecvResE[0], "U6", 5, acRecvDataE, aRecvData2[0], abRecvResE);
INCP(_e1, iVar8);
TON_2(IN := NOT U6\G20485.4, PT := T#5s);
_e2 := INCP(TON_2.Q, CntRecvErr2);
bRecvErrE := _e2;
(* network 16 *)
INC(abRecvResE[0] AND NOT abRecvResE[1], CntRecv2);
MOVE_E(abRecvResE[0] AND abRecvResE[1], acRecvDataE[1], ErrCodeRE);
END_PROGRAM

PROGRAM Ex_SOCRCVS
VAR
  bOpenReqC : BOOL;
  bOpenOkC : BOOL;
  bOpenErrC : BOOL;
  abOpenResC : ARRAY [0..1] OF BOOL;
  acOpenData : ARRAY [0..9] OF INT;
  bSendReqC : BOOL;
  bSendOkC : BOOL;
  bSendErrC : BOOL;
  abSendResC : ARRAY [0..1] OF BOOL;
  acSendDataC : ARRAY [0..1] OF INT;
  bRecvOkC : BOOL;
  bRecvErrC : BOOL;
  abRecvResC : ARRAY [0..1] OF BOOL;
  bCloseReq : BOOL;
  bCloseOkC : BOOL;
  bCloseErrC : BOOL;
  abCloseResC : ARRAY [0..1] OF BOOL;
  acCloseData : ARRAY [0..1] OF INT;
  CntSend1 : INT;
  CntSend2 : INT;
  CntRecv1 : INT;
  CntRecv2 : INT;
  Mov4INT_1 : Mov4INT;
  Mov8INT_1 : Mov8INT;
  acRdCtrl : ARRAY [0..9] OF INT;
  Mov4INT_2 : Mov4INT;
  bOpenReqE : BOOL;
  bOpenOkE : BOOL;
  bOpenErrE : BOOL;
  abOpenResE : ARRAY [0..1] OF BOOL;
  bSendErrE : BOOL;
  bSendOkE : BOOL;
  bSendReqE : BOOL;
  abSendResE : ARRAY [0..1] OF BOOL;
  abRecvResE : ARRAY [0..1] OF BOOL;
  bRecvErrE : BOOL;
  bRecvOkE : BOOL;
  abCloseResE : ARRAY [0..1] OF BOOL;
  bCloseErrE : BOOL;
  bCloseOkE : BOOL;
  acSendDataE : ARRAY [0..1] OF INT;
  acRecvDataC : ARRAY [0..1] OF INT;
  acRecvDataE : ARRAY [0..1] OF INT;
  Word2Bit8_1 : Word2Bit8;
  Word2Bit8_2 : Word2Bit8;
  Word2Bit8_3 : Word2Bit8;
  Word2Bit8_4 : Word2Bit8;
  Word2Bit8_5 : Word2Bit8;
  Word2Bit8_6 : Word2Bit8;
  ErrCodeSC : INT;
  ErrCodeSE : INT;
  Mov4INT_3 : Mov4INT;
  bChangeReqC : BOOL;
  Mov4INT_4 : Mov4INT;
  acCsetData : ARRAY [0..4] OF INT;
  TON_1 : TON;
  CntRecvErr1 : INT;
  CntRecvErr2 : INT;
  TON_2 : TON;
  ErrCodeRC : INT;
  ErrCodeRE : INT;
  bRecvFlag : BOOL;
END_VAR
(* structured ladder/FBD written out as ST: instructions are called as NAME(EN, inputs, outputs); _pN, _eN, _tN stand for wires *)
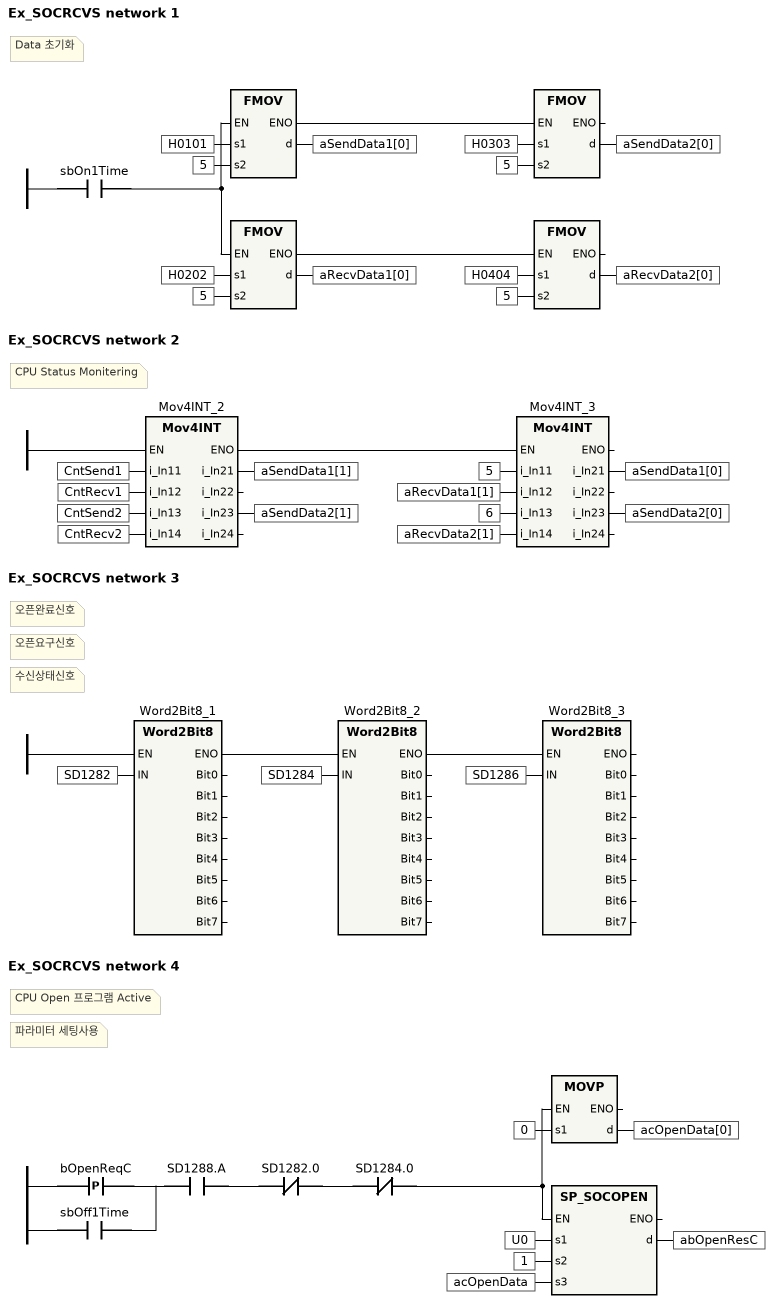
(* network 1 *)
(* Data 초기화 *)
_e1 := FMOV(sbOn1Time, H0101, 5, aSendData1[0]);
FMOV(_e1, H0303, 5, aSendData2[0]);
_e2 := FMOV(sbOn1Time, H0202, 5, aRecvData1[0]);
FMOV(_e2, H0404, 5, aRecvData2[0]);
(* network 2 *)
(* CPU Status Monitering *)
Mov4INT_2(EN := TRUE, i_In11 := CntSend1, i_In12 := CntRecv1, i_In13 := CntSend2, i_In14 := CntRecv2, i_In21 => aSendData1[1], i_In23 => aSendData2[1]);
Mov4INT_3(EN := Mov4INT_2.ENO, i_In11 := 5, i_In12 := aRecvData1[1], i_In13 := 6, i_In14 := aRecvData2[1], i_In21 => aSendData1[0], i_In23 => aSendData2[0]);
(* network 3 *)
(* 오픈완료신호 *)
(* 오픈요구신호 *)
(* 수신상태신호 *)
Word2Bit8_1(EN := TRUE, IN := SD1282);
Word2Bit8_2(EN := Word2Bit8_1.ENO, IN := SD1284);
Word2Bit8_3(EN := Word2Bit8_2.ENO, IN := SD1286);
(* network 4 *)
(* CPU Open 프로그램 Active *)
(* 파라미터 세팅사용 *)
_p1 := (((LDP(TRUE, bOpenReqC) OR sbOff1Time) AND SD1288.A) AND NOT SD1282.0) AND NOT SD1284.0;
MOVP(_p1, 0, acOpenData[0]);
SP_SOCOPEN(_p1, U0, 1, acOpenData, abOpenResC);
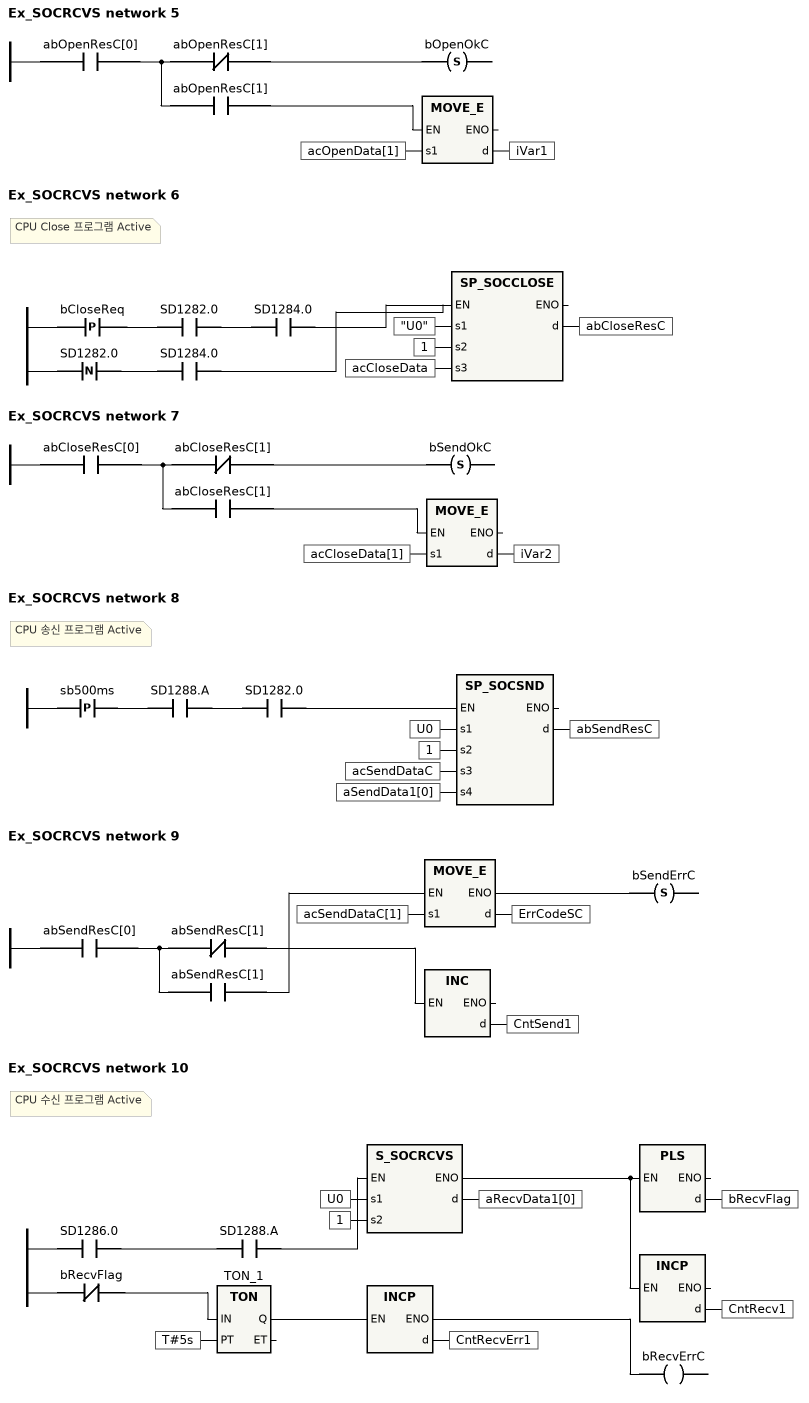
(* network 5 *)
SET(abOpenResC[0] AND NOT abOpenResC[1], bOpenOkC);
MOVE_E(abOpenResC[0] AND abOpenResC[1], acOpenData[1], iVar1);
(* network 6 *)
(* CPU Close 프로그램 Active *)
SP_SOCCLOSE((LDP(TRUE, bCloseReq) AND SD1282.0 AND SD1284.0) OR (LDF(TRUE, SD1282.0) AND SD1284.0), "U0", 1, acCloseData, abCloseResC);
(* network 7 *)
SET(abCloseResC[0] AND NOT abCloseResC[1], bSendOkC);
MOVE_E(abCloseResC[0] AND abCloseResC[1], acCloseData[1], iVar2);
(* network 8 *)
(* CPU 송신 프로그램 Active *)
SP_SOCSND(LDP(TRUE, sb500ms) AND SD1288.A AND SD1282.0, U0, 1, acSendDataC, aSendData1[0], abSendResC);
(* network 9 *)
INC(abSendResC[0] AND NOT abSendResC[1], CntSend1);
_e1 := MOVE_E(abSendResC[0] AND abSendResC[1], acSendDataC[1], ErrCodeSC);
SET(_e1, bSendErrC);
(* network 10 *)
(* CPU 수신 프로그램 Active *)
_e1 := S_SOCRCVS(SD1286.0 AND SD1288.A, U0, 1, aRecvData1[0]);
PLS(_e1, bRecvFlag);
INCP(_e1, CntRecv1);
TON_1(IN := NOT bRecvFlag, PT := T#5s);
_e2 := INCP(TON_1.Q, CntRecvErr1);
bRecvErrC := _e2;
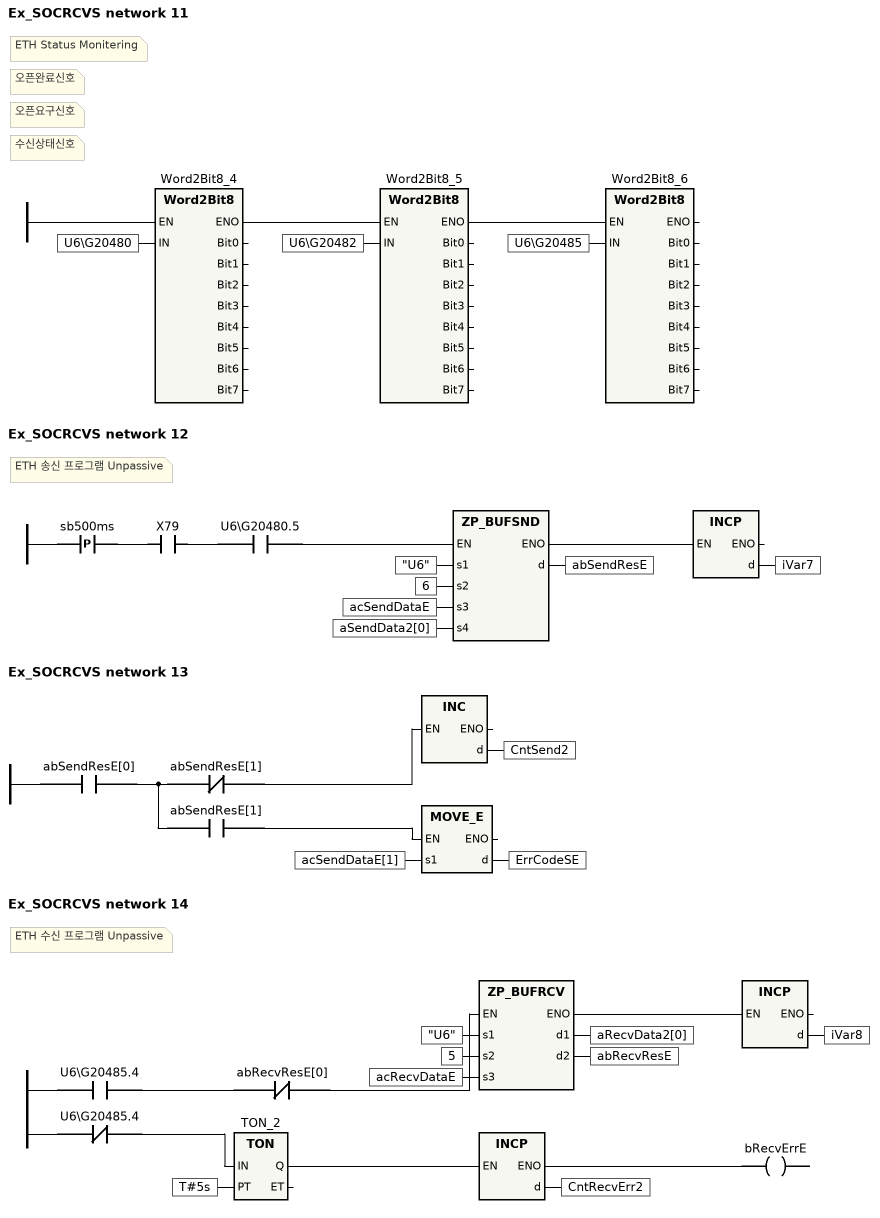
(* network 11 *)
(* ETH Status Monitering *)
(* 오픈완료신호 *)
(* 오픈요구신호 *)
(* 수신상태신호 *)
Word2Bit8_4(EN := TRUE, IN := U6\G20480);
Word2Bit8_5(EN := Word2Bit8_4.ENO, IN := U6\G20482);
Word2Bit8_6(EN := Word2Bit8_5.ENO, IN := U6\G20485);
(* network 12 *)
(* ETH 송신 프로그램 Unpassive *)
_e1 := ZP_BUFSND(LDP(TRUE, sb500ms) AND X79 AND U6\G20480.5, "U6", 6, acSendDataE, aSendData2[0], abSendResE);
INCP(_e1, iVar7);
(* network 13 *)
INC(abSendResE[0] AND NOT abSendResE[1], CntSend2);
MOVE_E(abSendResE[0] AND abSendResE[1], acSendDataE[1], ErrCodeSE);
(* network 14 *)
(* ETH 수신 프로그램 Unpassive *)
_e1 := ZP_BUFRCV(U6\G20485.4 AND NOT abRecvResE[0], "U6", 5, acRecvDataE, aRecvData2[0], abRecvResE);
INCP(_e1, iVar8);
TON_2(IN := NOT U6\G20485.4, PT := T#5s);
_e2 := INCP(TON_2.Q, CntRecvErr2);
bRecvErrE := _e2;
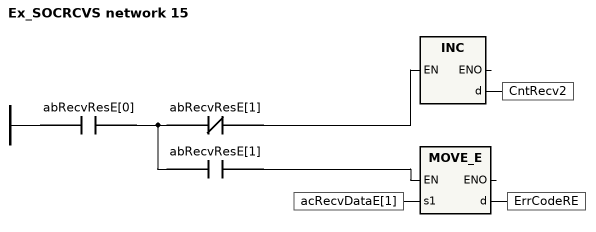
(* network 15 *)
INC(abRecvResE[0] AND NOT abRecvResE[1], CntRecv2);
MOVE_E(abRecvResE[0] AND abRecvResE[1], acRecvDataE[1], ErrCodeRE);
END_PROGRAM

PROGRAM Ex_SOCSND
VAR
  bOpenReqC : BOOL;
  bOpenOkC : BOOL;
  bOpenErrC : BOOL;
  abOpenResC : ARRAY [0..1] OF BOOL;
  acOpenData : ARRAY [0..9] OF INT;
  bSendReqC : BOOL;
  bSendOkC : BOOL;
  bSendErrC : BOOL;
  abSendResC : ARRAY [0..1] OF BOOL;
  acSendDataC : ARRAY [0..1] OF INT;
  bRecvOkC : BOOL;
  bRecvErrC : BOOL;
  abRecvResC : ARRAY [0..1] OF BOOL;
  bCloseReq : BOOL;
  bCloseOkC : BOOL;
  bCloseErrC : BOOL;
  abCloseResC : ARRAY [0..1] OF BOOL;
  acCloseData : ARRAY [0..1] OF INT;
  CntSend1 : INT;
  CntSend2 : INT;
  CntRecv1 : INT;
  CntRecv2 : INT;
  Mov4INT_1 : Mov4INT;
  Mov8INT_1 : Mov8INT;
  acRdCtrl : ARRAY [0..9] OF INT;
  Mov4INT_2 : Mov4INT;
  bOpenReqE : BOOL;
  bOpenOkE : BOOL;
  bOpenErrE : BOOL;
  abOpenResE : ARRAY [0..1] OF BOOL;
  bSendErrE : BOOL;
  bSendOkE : BOOL;
  bSendReqE : BOOL;
  abSendResE : ARRAY [0..1] OF BOOL;
  abRecvResE : ARRAY [0..1] OF BOOL;
  bRecvErrE : BOOL;
  bRecvOkE : BOOL;
  abCloseResE : ARRAY [0..1] OF BOOL;
  bCloseErrE : BOOL;
  bCloseOkE : BOOL;
  acSendDataE : ARRAY [0..1] OF INT;
  acRecvDataC : ARRAY [0..1] OF INT;
  acRecvDataE : ARRAY [0..1] OF INT;
  Word2Bit8_1 : Word2Bit8;
  Word2Bit8_2 : Word2Bit8;
  Word2Bit8_3 : Word2Bit8;
  Word2Bit8_4 : Word2Bit8;
  Word2Bit8_5 : Word2Bit8;
  Word2Bit8_6 : Word2Bit8;
  ErrCodeSC : INT;
  ErrCodeSE : INT;
  Mov4INT_3 : Mov4INT;
  bChangeReqC : BOOL;
  Mov4INT_4 : Mov4INT;
  acCsetData : ARRAY [0..4] OF INT;
  TON_1 : TON;
  CntRecvErr1 : INT;
  CntRecvErr2 : INT;
  TON_2 : TON;
  ErrCodeRC : INT;
  ErrCodeRE : INT;
  Mov4INT_5 : Mov4INT;
END_VAR
(* structured ladder/FBD written out as ST: instructions are called as NAME(EN, inputs, outputs); _pN, _eN, _tN stand for wires *)
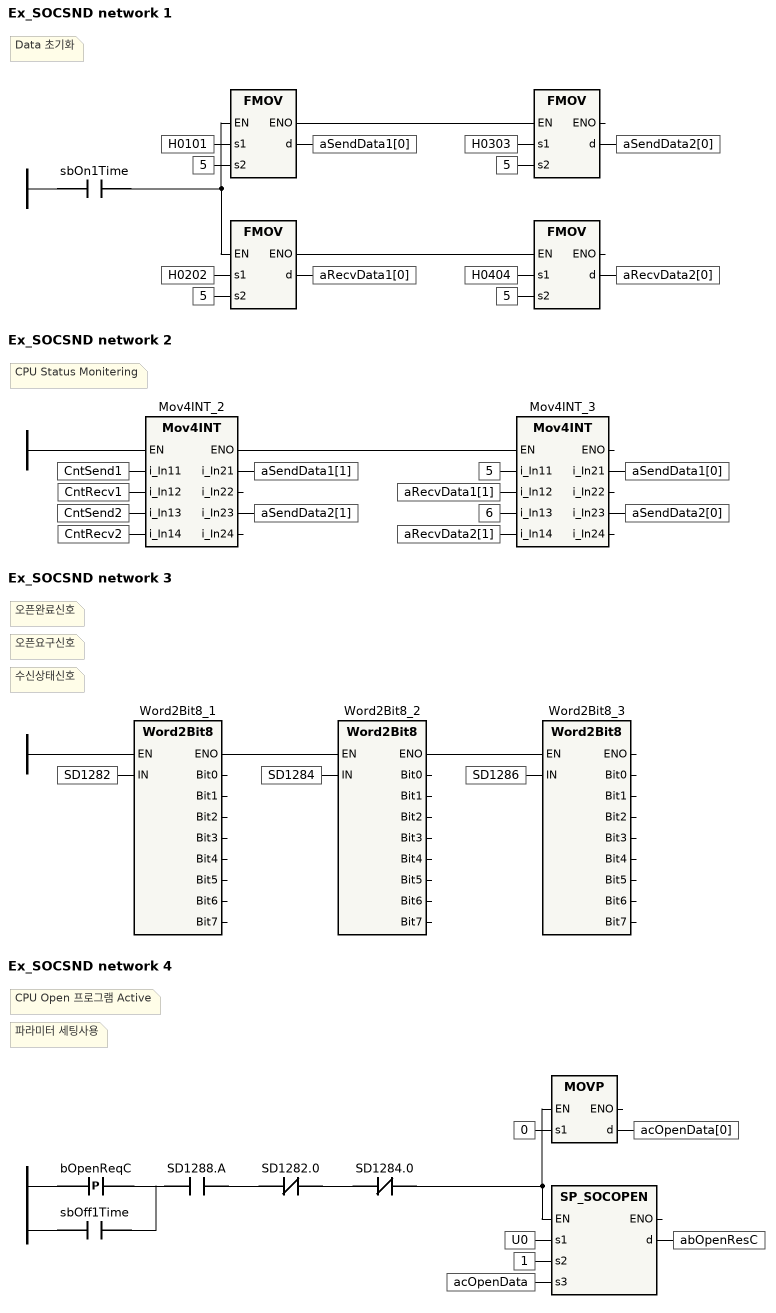
(* network 1 *)
(* Data 초기화 *)
_e1 := FMOV(sbOn1Time, H0101, 5, aSendData1[0]);
FMOV(_e1, H0303, 5, aSendData2[0]);
_e2 := FMOV(sbOn1Time, H0202, 5, aRecvData1[0]);
FMOV(_e2, H0404, 5, aRecvData2[0]);
(* network 2 *)
(* CPU Status Monitering *)
Mov4INT_2(EN := TRUE, i_In11 := CntSend1, i_In12 := CntRecv1, i_In13 := CntSend2, i_In14 := CntRecv2, i_In21 => aSendData1[1], i_In23 => aSendData2[1]);
Mov4INT_3(EN := Mov4INT_2.ENO, i_In11 := 5, i_In12 := aRecvData1[1], i_In13 := 6, i_In14 := aRecvData2[1], i_In21 => aSendData1[0], i_In23 => aSendData2[0]);
(* network 3 *)
(* 오픈완료신호 *)
(* 오픈요구신호 *)
(* 수신상태신호 *)
Word2Bit8_1(EN := TRUE, IN := SD1282);
Word2Bit8_2(EN := Word2Bit8_1.ENO, IN := SD1284);
Word2Bit8_3(EN := Word2Bit8_2.ENO, IN := SD1286);
(* network 4 *)
(* CPU Open 프로그램 Active *)
(* 파라미터 세팅사용 *)
_p1 := (((LDP(TRUE, bOpenReqC) OR sbOff1Time) AND SD1288.A) AND NOT SD1282.0) AND NOT SD1284.0;
MOVP(_p1, 0, acOpenData[0]);
SP_SOCOPEN(_p1, U0, 1, acOpenData, abOpenResC);
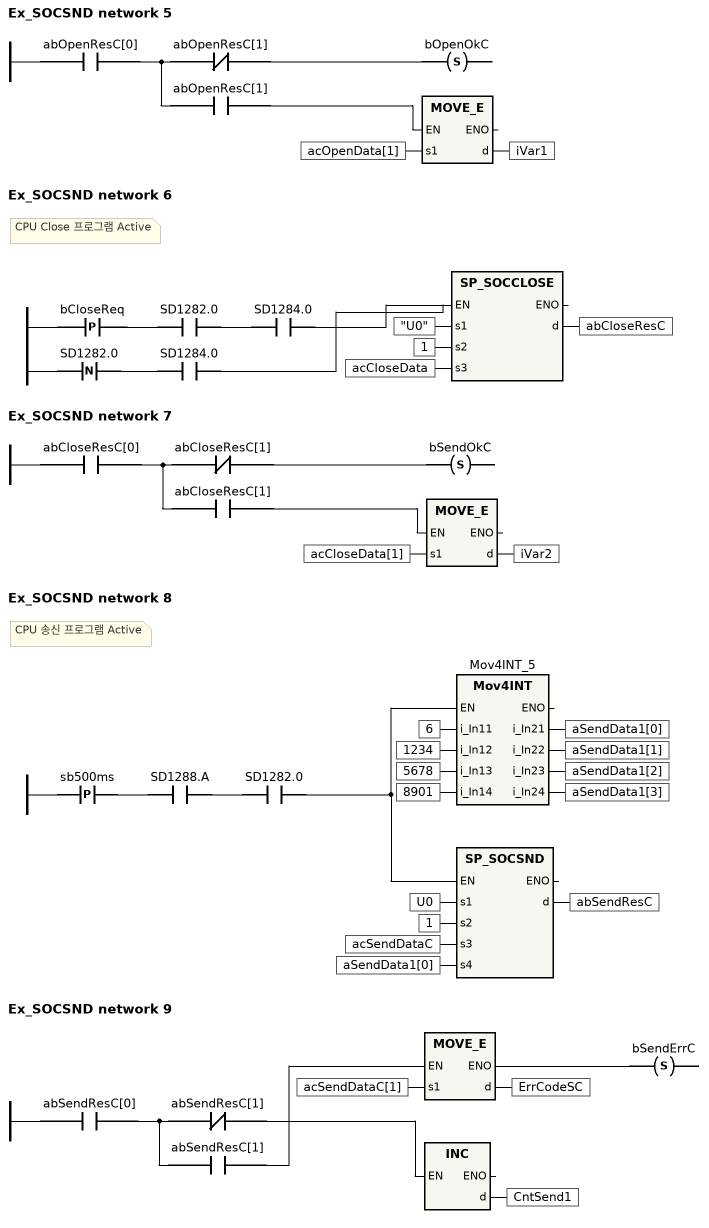
(* network 5 *)
SET(abOpenResC[0] AND NOT abOpenResC[1], bOpenOkC);
MOVE_E(abOpenResC[0] AND abOpenResC[1], acOpenData[1], iVar1);
(* network 6 *)
(* CPU Close 프로그램 Active *)
SP_SOCCLOSE((LDP(TRUE, bCloseReq) AND SD1282.0 AND SD1284.0) OR (LDF(TRUE, SD1282.0) AND SD1284.0), "U0", 1, acCloseData, abCloseResC);
(* network 7 *)
SET(abCloseResC[0] AND NOT abCloseResC[1], bSendOkC);
MOVE_E(abCloseResC[0] AND abCloseResC[1], acCloseData[1], iVar2);
(* network 8 *)
(* CPU 송신 프로그램 Active *)
_p1 := LDP(TRUE, sb500ms) AND SD1288.A AND SD1282.0;
Mov4INT_5(EN := _p1, i_In11 := 6, i_In12 := 1234, i_In13 := 5678, i_In14 := 8901, i_In21 => aSendData1[0], i_In22 => aSendData1[1], i_In23 => aSendData1[2], i_In24 => aSendData1[3]);
SP_SOCSND(_p1, U0, 1, acSendDataC, aSendData1[0], abSendResC);
(* network 9 *)
INC(abSendResC[0] AND NOT abSendResC[1], CntSend1);
_e1 := MOVE_E(abSendResC[0] AND abSendResC[1], acSendDataC[1], ErrCodeSC);
SET(_e1, bSendErrC);
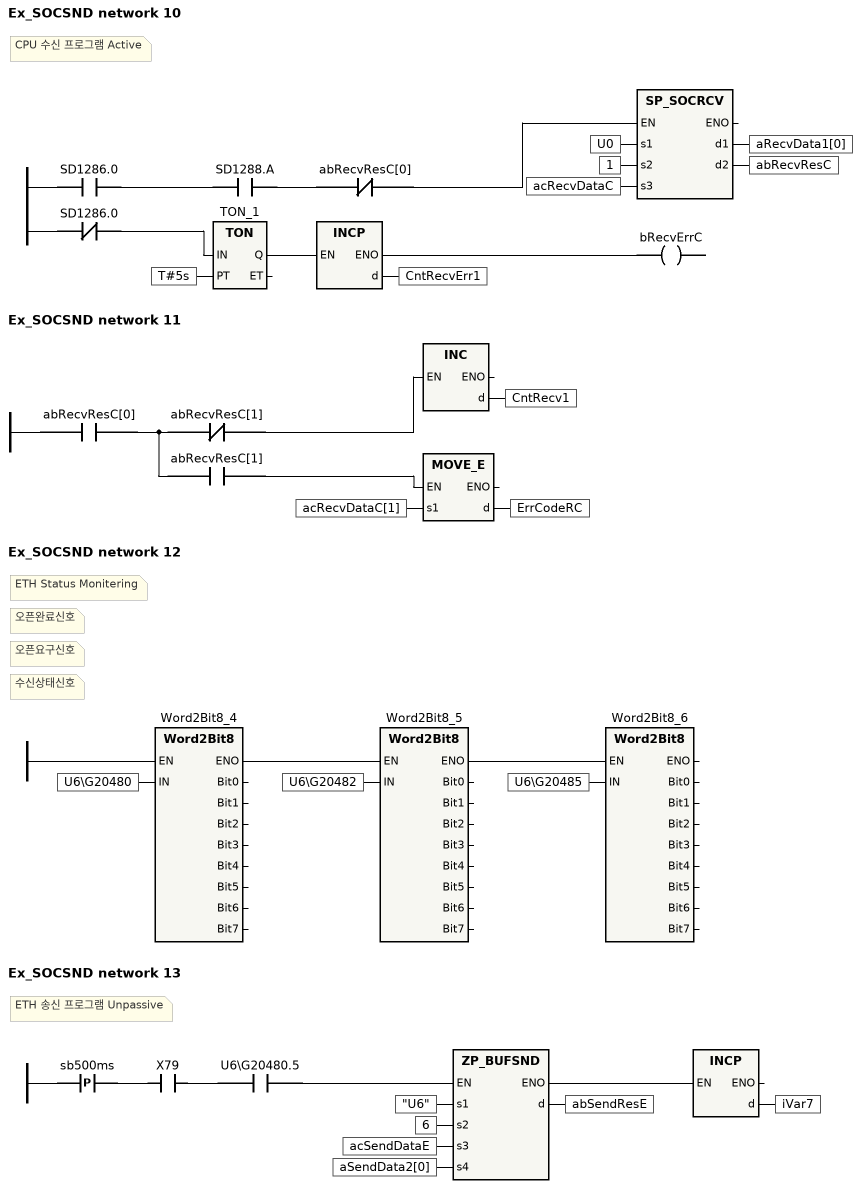
(* network 10 *)
(* CPU 수신 프로그램 Active *)
SP_SOCRCV(SD1286.0 AND SD1288.A AND NOT abRecvResC[0], U0, 1, acRecvDataC, aRecvData1[0], abRecvResC);
TON_1(IN := NOT SD1286.0, PT := T#5s);
_e1 := INCP(TON_1.Q, CntRecvErr1);
bRecvErrC := _e1;
(* network 11 *)
INC(abRecvResC[0] AND NOT abRecvResC[1], CntRecv1);
MOVE_E(abRecvResC[0] AND abRecvResC[1], acRecvDataC[1], ErrCodeRC);
(* network 12 *)
(* ETH Status Monitering *)
(* 오픈완료신호 *)
(* 오픈요구신호 *)
(* 수신상태신호 *)
Word2Bit8_4(EN := TRUE, IN := U6\G20480);
Word2Bit8_5(EN := Word2Bit8_4.ENO, IN := U6\G20482);
Word2Bit8_6(EN := Word2Bit8_5.ENO, IN := U6\G20485);
(* network 13 *)
(* ETH 송신 프로그램 Unpassive *)
_e1 := ZP_BUFSND(LDP(TRUE, sb500ms) AND X79 AND U6\G20480.5, "U6", 6, acSendDataE, aSendData2[0], abSendResE);
INCP(_e1, iVar7);
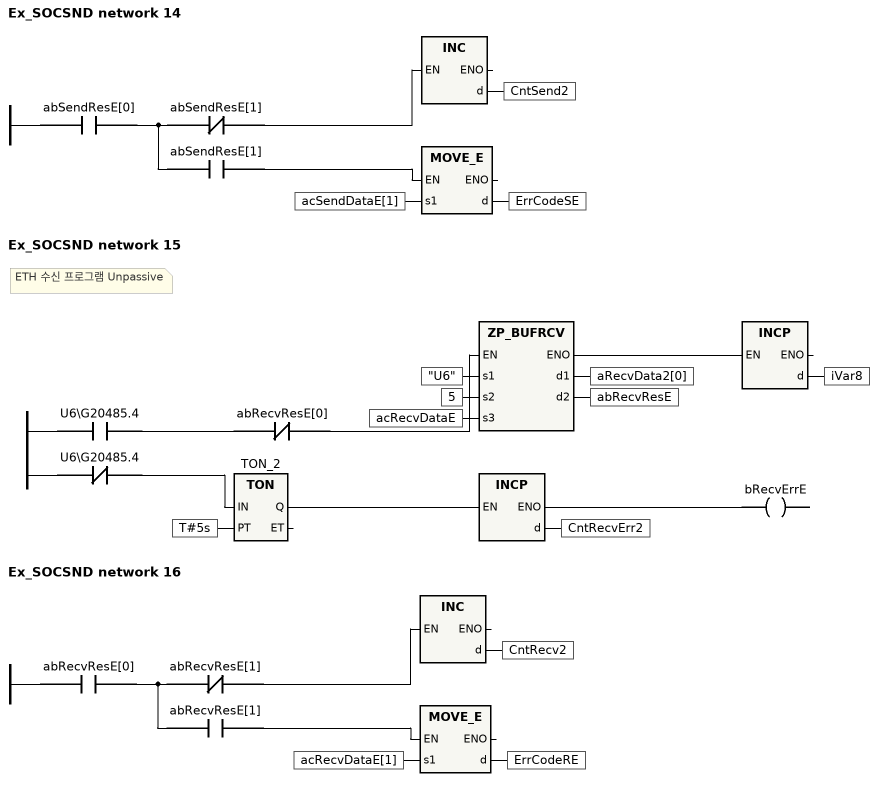
(* network 14 *)
INC(abSendResE[0] AND NOT abSendResE[1], CntSend2);
MOVE_E(abSendResE[0] AND abSendResE[1], acSendDataE[1], ErrCodeSE);
(* network 15 *)
(* ETH 수신 프로그램 Unpassive *)
_e1 := ZP_BUFRCV(U6\G20485.4 AND NOT abRecvResE[0], "U6", 5, acRecvDataE, aRecvData2[0], abRecvResE);
INCP(_e1, iVar8);
TON_2(IN := NOT U6\G20485.4, PT := T#5s);
_e2 := INCP(TON_2.Q, CntRecvErr2);
bRecvErrE := _e2;
(* network 16 *)
INC(abRecvResE[0] AND NOT abRecvResE[1], CntRecv2);
MOVE_E(abRecvResE[0] AND abRecvResE[1], acRecvDataE[1], ErrCodeRE);
END_PROGRAM

PROGRAM Ex_SOCCINF
VAR
  bOpenReqC : BOOL;
  bOpenOkC : BOOL;
  bOpenErrC : BOOL;
  abOpenResC : ARRAY [0..1] OF BOOL;
  acOpenData : ARRAY [0..9] OF INT;
  acInfoData1 : ARRAY [0..1] OF INT;
  bOpenReqE : BOOL;
  bOpenOkE : BOOL;
  bOpenErrE : BOOL;
  abOpenResE : ARRAY [0..1] OF BOOL;
  bInfoReq : BOOL;
  acInfoData2 : ARRAY [0..1] OF INT;
  aInfo1 : ARRAY [0..4] OF INT;
  aInfo2 : ARRAY [0..4] OF INT;
  Mov8INT_1 : Mov8INT;
  Mov8INT_2 : Mov8INT;
END_VAR
(* structured ladder/FBD written out as ST: instructions are called as NAME(EN, inputs, outputs); _pN, _eN, _tN stand for wires *)
